LIN {X 0,Y 523.515,Z 542.317,A -85,B 0,C 180,E1 -4776.742,E2 -4776.742} C_VEL
LIN {X 0,Y 523.666,Z 535.608,A -85,B 0,C 180,E1 -4777.907,E2 -4777.907} C_VEL
LIN {X 0,Y 523.85,Z 527.307,A -85,B 0,C 180,E1 -4779.07,E2 -4779.07} C_VEL
LIN {X 0,Y 524.067,Z 518.801,A -85,B 0,C 180,E1 -4780.04,E2 -4780.04} C_VEL
LIN {X 0,Y 524.36,Z 508.293,A -85,B 0,C 180,E1 -4781.011,E2 -4781.011} C_VEL
LIN {X 0,Y 524.681,Z 496.847,A -85,B 0,C 180,E1 -4781.859,E2 -4781.859} C_VEL
LIN {X 0,Y 524.929,Z 486.505,A -85,B 0,C 180,E1 -4782.468,E2 -4782.468} C_VEL
LIN {X 0,Y 525.138,Z 474.81,A -85,B 0,C 180,E1 -4783.003,E2 -4783.003} C_VEL
LIN {X 0,Y 525.391,Z 461.34,A -85,B 0,C 180,E1 -4783.44,E2 -4783.44} C_VEL
LIN {X 0,Y 525.559,Z 448.003,A -85,B 0,C 180,E1 -4783.706,E2 -4783.706} C_VEL
LIN {X 0,Y 525.857,Z 355.901,A -85,B 0,C 180,E1 -4784.97,E2 -4784.97} C_VEL
LIN {X 0,Y 524.303,Z 345.51,A -85,B 0,C 180,E1 -4785.176,E2 -4785.176} C_VEL
LIN {X 0,Y 524.737,Z 323.457,A -85,B 0,C 180,E1 -4788.528,E2 -4788.528} C_VEL
LIN {X 0,Y 525.117,Z 304.861,A -85,B 0,C 180,E1 -4791.39,E2 -4791.39} C_VEL
LIN {X 0,Y 525.357,Z 292.969,A -85,B 0,C 180,E1 -4793.243,E2 -4793.243} C_VEL
LIN {X 0,Y 523.98,Z 285.215,A -85,B 0,C 180,E1 -4794.569,E2 -4794.569} C_VEL
LIN {X 0,Y 523.949,Z 285.218,A -85,B 0,C 180,E1 -4797.133,E2 -4797.133} C_VEL
LIN {X 0,Y 523.944,Z 285.223,A -85,B 0,C 180,E1 -4799.756,E2 -4799.756} C_VEL
LIN {X 0,Y 523.935,Z 285.221,A -85,B 0,C 180,E1 -4802.449,E2 -4802.449} C_VEL
LIN {X 0,Y 523.921,Z 285.218,A -85,B 0,C 180,E1 -4805.227,E2 -4805.227} C_VEL
LIN {X 0,Y 523.917,Z 285.225,A -85,B 0,C 180,E1 -4808.102,E2 -4808.102} C_VEL
LIN {X 0,Y 523.94,Z 285.217,A -85,B 0,C 180,E1 -4811.092,E2 -4811.092} C_VEL
LIN {X 0,Y 523.931,Z 285.221,A -85,B 0,C 180,E1 -4814.229,E2 -4814.229} C_VEL
LIN {X 0,Y 523.917,Z 285.225,A -85,B 0,C 180,E1 -4816.832,E2 -4816.832} C_VEL
LIN {X 0,Y 523.939,Z 285.221,A -85,B 0,C 180,E1 -4818.907,E2 -4818.907} C_VEL
LIN {X 0,Y 523.915,Z 285.218,A -85,B 0,C 180,E1 -4821.898,E2 -4821.898} C_VEL
LIN {X 0,Y 523.924,Z 285.226,A -85,B 0,C 180,E1 -4824.911,E2 -4824.911} C_VEL
LIN {X 0,Y 523.934,Z 285.217,A -85,B 0,C 180,E1 -4827.679,E2 -4827.679} C_VEL
LIN {X 0,Y 523.953,Z 285.216,A -85,B 0,C 180,E1 -4830.676,E2 -4830.676} C_VEL
LIN {X 0,Y 523.973,Z 285.213,A -85,B 0,C 180,E1 -4833.728,E2 -4833.728} C_VEL
LIN {X 0,Y 523.925,Z 285.216,A -85,B 0,C 180,E1 -4836.27,E2 -4836.27} C_VEL
LIN {X 0,Y 523.945,Z 285.216,A -85,B 0,C 180,E1 -4838.766,E2 -4838.766} C_VEL
LIN {X 0,Y 523.95,Z 285.22,A -85,B 0,C 180,E1 -4841.221,E2 -4841.221} C_VEL
LIN {X 0,Y 523.936,Z 285.222,A -85,B 0,C 180,E1 -4843.639,E2 -4843.639} C_VEL
LIN {X 0,Y 523.942,Z 285.216,A -85,B 0,C 180,E1 -4846.028,E2 -4846.028} C_VEL
LIN {X 0,Y 524.011,Z 285.206,A -85,B 0,C 180,E1 -4848.394,E2 -4848.394} C_VEL
LIN {X 0,Y 524.001,Z 285.211,A -85,B 0,C 180,E1 -4851.516,E2 -4851.516} C_VEL
LIN {X 0,Y 524.079,Z 285.195,A -85,B 0,C 180,E1 -4854.614,E2 -4854.614} C_VEL
LIN {X 0,Y 524.11,Z 285.198,A -85,B 0,C 180,E1 -4857.694,E2 -4857.694} C_VEL
LIN {X 0,Y 524.12,Z 285.192,A -85,B 0,C 180,E1 -4860.768,E2 -4860.768} C_VEL
LIN {X 0,Y 524.07,Z 285.195,A -85,B 0,C 180,E1 -4863.075,E2 -4863.075} C_VEL
LIN {X 0,Y 524.035,Z 285.211,A -85,B 0,C 180,E1 -4866.159,E2 -4866.159} C_VEL
LIN {X 0,Y 524.001,Z 285.213,A -85,B 0,C 180,E1 -4868.484,E2 -4868.484} C_VEL
LIN {X 0,Y 524,Z 285.207,A -85,B 0,C 180,E1 -4871.739,E2 -4871.739} C_VEL
LIN {X 0,Y 523.992,Z 285.21,A -85,B 0,C 180,E1 -4875.053,E2 -4875.053} C_VEL
LIN {X 0,Y 523.962,Z 285.213,A -85,B 0,C 180,E1 -4877.969,E2 -4877.969} C_VEL
LIN {X 0,Y 523.97,Z 285.217,A -85,B 0,C 180,E1 -4880.41,E2 -4880.41} C_VEL
LIN {X 0,Y 523.915,Z 285.225,A -85,B 0,C 180,E1 -4882.893,E2 -4882.893} C_VEL
LIN {X 0,Y 523.951,Z 285.215,A -85,B 0,C 180,E1 -4885.419,E2 -4885.419} C_VEL
LIN {X 0,Y 523.966,Z 285.21,A -85,B 0,C 180,E1 -4887.999,E2 -4887.999} C_VEL
LIN {X 0,Y 523.943,Z 285.222,A -85,B 0,C 180,E1 -4890.855,E2 -4890.855} C_VEL
LIN {X 0,Y 523.957,Z 285.213,A -85,B 0,C 180,E1 -4893.735,E2 -4893.735} C_VEL
LIN {X 0,Y 523.902,Z 285.22,A -85,B 0,C 180,E1 -4896.401,E2 -4896.401} C_VEL
LIN {X 0,Y 523.919,Z 285.225,A -85,B 0,C 180,E1 -4899.085,E2 -4899.085} C_VEL
LIN {X 0,Y 523.951,Z 285.214,A -85,B 0,C 180,E1 -4902.119,E2 -4902.119} C_VEL
LIN {X 0,Y 523.941,Z 285.223,A -85,B 0,C 180,E1 -4905.31,E2 -4905.31} C_VEL
LIN {X 0,Y 523.914,Z 285.22,A -85,B 0,C 180,E1 -4906.905,E2 -4906.905} C_VEL
LIN {X 0,Y 523.25,Z 285.311,A -85,B 0,C 180,E1 -4907.546,E2 -4907.546} C_VEL
LIN {X 0,Y 520.41,Z 285.663,A -85,B 0,C 180,E1 -4908.588,E2 -4908.588} C_VEL
LIN {X 0,Y 518.006,Z 285.962,A -85,B 0,C 180,E1 -4909.427,E2 -4909.427} C_VEL
LIN {X 0,Y 516.969,Z 286.088,A -85,B 0,C 180,E1 -4910.075,E2 -4910.075} C_VEL
LIN {X 0,Y 516.881,Z 286.097,A -85,B 0,C 180,E1 -4910.294,E2 -4910.294} C_VEL
LIN {X 0,Y 516.877,Z 286.1,A -85,B 0,C 180,E1 -4913.343,E2 -4913.343} C_VEL
LIN {X 0,Y 516.907,Z 286.098,A -85,B 0,C 180,E1 -4916.121,E2 -4916.121} C_VEL
LIN {X 0,Y 516.892,Z 286.097,A -85,B 0,C 180,E1 -4918.936,E2 -4918.936} C_VEL
LIN {X 0,Y 516.971,Z 286.237,A -85,B 0,C 180,E1 -4920.438,E2 -4920.438} C_VEL
LIN {X 0,Y 517.368,Z 291.344,A -85,B 0,C 180,E1 -4921.39,E2 -4921.39} C_VEL
LIN {X 0,Y 517.217,Z 308.839,A -85,B 0,C 180,E1 -4924.604,E2 -4924.604} C_VEL
LIN {X 0,Y 517.184,Z 309.29,A -85,B 0,C 180,E1 -4924.685,E2 -4924.685} C_VEL
LIN {X 0,Y 519.153,Z 320.399,A -85,B 0,C 180,E1 -4924.906,E2 -4924.906} C_VEL
LIN {X 0,Y 518.582,Z 416.061,A -85,B 0,C 180,E1 -4926.249,E2 -4926.249} C_VEL
LIN {X 0,Y 518.424,Z 429.105,A -85,B 0,C 180,E1 -4926.586,E2 -4926.586} C_VEL
LIN {X 0,Y 518.222,Z 441.25,A -85,B 0,C 180,E1 -4927.051,E2 -4927.051} C_VEL
LIN {X 0,Y 517.957,Z 453.258,A -85,B 0,C 180,E1 -4927.671,E2 -4927.671} C_VEL
LIN {X 0,Y 517.642,Z 464.025,A -85,B 0,C 180,E1 -4928.391,E2 -4928.391} C_VEL
LIN {X 0,Y 517.359,Z 475.056,A -85,B 0,C 180,E1 -4929.317,E2 -4929.317} C_VEL
LIN {X 0,Y 517.034,Z 484.878,A -85,B 0,C 180,E1 -4930.341,E2 -4930.341} C_VEL
LIN {X 0,Y 516.799,Z 494.224,A -85,B 0,C 180,E1 -4931.568,E2 -4931.568} C_VEL
LIN {X 0,Y 516.605,Z 501.678,A -85,B 0,C 180,E1 -4932.789,E2 -4932.789} C_VEL
LIN {X 0,Y 516.447,Z 506.653,A -85,B 0,C 180,E1 -4933.801,E2 -4933.801} C_VEL
LIN {X 0,Y 516.405,Z 511.668,A -85,B 0,C 180,E1 -4935.077,E2 -4935.077} C_VEL
LIN {X 0,Y 516.31,Z 515.051,A -85,B 0,C 180,E1 -4936.219,E2 -4936.219} C_VEL
LIN {X 0,Y 516.23,Z 517.598,A -85,B 0,C 180,E1 -4937.418,E2 -4937.418} C_VEL
LIN {X 0,Y 516.282,Z 519.102,A -85,B 0,C 180,E1 -4938.555,E2 -4938.555} C_VEL
LIN {X 0,Y 516.238,Z 519.799,A -85,B 0,C 180,E1 -4939.806,E2 -4939.806} C_VEL
LIN {X 0,Y 516.176,Z 519.736,A -85,B 0,C 180,E1 -4940.596,E2 -4940.596} C_VEL
LIN {X 0,Y 516.213,Z 519.25,A -85,B 0,C 180,E1 -4941.387,E2 -4941.387} C_VEL
LIN {X 0,Y 516.267,Z 518.344,A -85,B 0,C 180,E1 -4942.176,E2 -4942.176} C_VEL
LIN {X 0,Y 516.37,Z 515.929,A -85,B 0,C 180,E1 -4943.494,E2 -4943.494} C_VEL
LIN {X 0,Y 516.315,Z 511.958,A -85,B 0,C 180,E1 -4944.924,E2 -4944.924} C_VEL
LIN {X 0,Y 516.425,Z 507.49,A -85,B 0,C 180,E1 -4946.098,E2 -4946.098} C_VEL
LIN {X 0,Y 516.568,Z 500.737,A -85,B 0,C 180,E1 -4947.465,E2 -4947.465} C_VEL
LIN {X 0,Y 516.788,Z 493.426,A -85,B 0,C 180,E1 -4948.636,E2 -4948.636} C_VEL
LIN {X 0,Y 517.068,Z 484.361,A -85,B 0,C 180,E1 -4949.805,E2 -4949.805} C_VEL
LIN {X 0,Y 517.273,Z 473.947,A -85,B 0,C 180,E1 -4950.875,E2 -4950.875} C_VEL
LIN {X 0,Y 517.65,Z 463.329,A -85,B 0,C 180,E1 -4951.75,E2 -4951.75} C_VEL
LIN {X 0,Y 517.952,Z 453.041,A -85,B 0,C 180,E1 -4952.43,E2 -4952.43} C_VEL
LIN {X 0,Y 518.208,Z 440.744,A -85,B 0,C 180,E1 -4953.061,E2 -4953.061} C_VEL
LIN {X 0,Y 518.409,Z 427.821,A -85,B 0,C 180,E1 -4953.546,E2 -4953.546} C_VEL
LIN {X 0,Y 518.626,Z 414.887,A -85,B 0,C 180,E1 -4953.86,E2 -4953.86} C_VEL
LIN {X 0,Y 519.096,Z 319.758,A -85,B 0,C 180,E1 -4955.194,E2 -4955.194} C_VEL
LIN {X 0,Y 517.207,Z 309.344,A -85,B 0,C 180,E1 -4955.409,E2 -4955.409} C_VEL
LIN {X 0,Y 517.397,Z 294.542,A -85,B 0,C 180,E1 -4958.199,E2 -4958.199} C_VEL
LIN {X 0,Y 517.281,Z 288.307,A -85,B 0,C 180,E1 -4959.383,E2 -4959.383} C_VEL
LIN {X 0,Y 516.903,Z 286.101,A -85,B 0,C 180,E1 -4959.834,E2 -4959.834} C_VEL
LIN {X 0,Y 516.898,Z 286.099,A -85,B 0,C 180,E1 -4962.564,E2 -4962.564} C_VEL
LIN {X 0,Y 516.883,Z 286.096,A -85,B 0,C 180,E1 -4965.779,E2 -4965.779} C_VEL
LIN {X 0,Y 516.87,Z 286.102,A -85,B 0,C 180,E1 -4968.223,E2 -4968.223} C_VEL
LIN {X 0,Y 516.9,Z 286.098,A -85,B 0,C 180,E1 -4970.701,E2 -4970.701} C_VEL
LIN {X 0,Y 516.854,Z 286.098,A -85,B 0,C 180,E1 -4973.223,E2 -4973.223} C_VEL
LIN {X 0,Y 516.865,Z 286.099,A -85,B 0,C 180,E1 -4976.178,E2 -4976.178} C_VEL
LIN {X 0,Y 516.899,Z 286.093,A -85,B 0,C 180,E1 -4979.305,E2 -4979.305} C_VEL
LIN {X 0,Y 516.887,Z 286.099,A -85,B 0,C 180,E1 -4982.542,E2 -4982.542} C_VEL
LIN {X 0,Y 516.86,Z 286.099,A -85,B 0,C 180,E1 -4985.329,E2 -4985.329} C_VEL
LIN {X 0,Y 516.873,Z 286.095,A -85,B 0,C 180,E1 -4987.942,E2 -4987.942} C_VEL
LIN {X 0,Y 516.848,Z 286.104,A -85,B 0,C 180,E1 -4990.744,E2 -4990.744} C_VEL
LIN {X 0,Y 516.875,Z 286.095,A -85,B 0,C 180,E1 -4993.903,E2 -4993.903} C_VEL
LIN {X 0,Y 516.874,Z 286.095,A -85,B 0,C 180,E1 -4996.107,E2 -4996.107} C_VEL
LIN {X 0,Y 516.873,Z 286.105,A -85,B 0,C 180,E1 -4999.257,E2 -4999.257} C_VEL
LIN {X 0,Y 516.855,Z 286.097,A -85,B 0,C 180,E1 -5002.273,E2 -5002.273} C_VEL
LIN {X 0,Y 516.875,Z 286.101,A -85,B 0,C 180,E1 -5005.175,E2 -5005.175} C_VEL
LIN {X 0,Y 516.865,Z 286.098,A -85,B 0,C 180,E1 -5007.975,E2 -5007.975} C_VEL
LIN {X 0,Y 516.912,Z 286.09,A -85,B 0,C 180,E1 -5010.695,E2 -5010.695} C_VEL
LIN {X 0,Y 516.931,Z 286.095,A -85,B 0,C 180,E1 -5013.804,E2 -5013.804} C_VEL
LIN {X 0,Y 516.851,Z 286.098,A -85,B 0,C 180,E1 -5016.776,E2 -5016.776} C_VEL
LIN {X 0,Y 516.93,Z 286.097,A -85,B 0,C 180,E1 -5019.731,E2 -5019.731} C_VEL
LIN {X 0,Y 516.92,Z 286.09,A -85,B 0,C 180,E1 -5022.596,E2 -5022.596} C_VEL
LIN {X 0,Y 516.931,Z 286.088,A -85,B 0,C 180,E1 -5025.03,E2 -5025.03} C_VEL
LIN {X 0,Y 516.956,Z 286.091,A -85,B 0,C 180,E1 -5028.234,E2 -5028.234} C_VEL
LIN {X 0,Y 516.959,Z 286.085,A -85,B 0,C 180,E1 -5031.4,E2 -5031.4} C_VEL
LIN {X 0,Y 517.016,Z 286.081,A -85,B 0,C 180,E1 -5034.54,E2 -5034.54} C_VEL
LIN {X 0,Y 517.073,Z 286.072,A -85,B 0,C 180,E1 -5037.663,E2 -5037.663} C_VEL
LIN {X 0,Y 517.086,Z 286.072,A -85,B 0,C 180,E1 -5040.779,E2 -5040.779} C_VEL
LIN {X 0,Y 517.006,Z 286.079,A -85,B 0,C 180,E1 -5043.117,E2 -5043.117} C_VEL
LIN {X 0,Y 517,Z 286.085,A -85,B 0,C 180,E1 -5046.243,E2 -5046.243} C_VEL
LIN {X 0,Y 516.949,Z 286.086,A -85,B 0,C 180,E1 -5049.389,E2 -5049.389} C_VEL
LIN {X 0,Y 516.949,Z 286.086,A -85,B 0,C 180,E1 -5051.81,E2 -5051.81} C_VEL
LIN {X 0,Y 516.938,Z 286.09,A -85,B 0,C 180,E1 -5055.148,E2 -5055.148} C_VEL
LIN {X 0,Y 516.917,Z 286.091,A -85,B 0,C 180,E1 -5058.223,E2 -5058.223} C_VEL
LIN {X 0,Y 516.904,Z 286.098,A -85,B 0,C 180,E1 -5060.702,E2 -5060.702} C_VEL
LIN {X 0,Y 516.904,Z 286.091,A -85,B 0,C 180,E1 -5064.073,E2 -5064.073} C_VEL
LIN {X 0,Y 516.922,Z 286.093,A -85,B 0,C 180,E1 -5066.658,E2 -5066.658} C_VEL
LIN {X 0,Y 516.913,Z 286.093,A -85,B 0,C 180,E1 -5069.526,E2 -5069.526} C_VEL
LIN {X 0,Y 516.894,Z 286.094,A -85,B 0,C 180,E1 -5072.545,E2 -5072.545} C_VEL
LIN {X 0,Y 516.873,Z 286.104,A -85,B 0,C 180,E1 -5075.333,E2 -5075.333} C_VEL
LIN {X 0,Y 516.879,Z 286.096,A -85,B 0,C 180,E1 -5077.944,E2 -5077.944} C_VEL
LIN {X 0,Y 516.881,Z 286.095,A -85,B 0,C 180,E1 -5080.742,E2 -5080.742} C_VEL
LIN {X 0,Y 516.9,Z 286.093,A -85,B 0,C 180,E1 -5082.83,E2 -5082.83} C_VEL
LIN {X 0,Y 516.919,Z 286.092,A -85,B 0,C 180,E1 -5085.011,E2 -5085.011} C_VEL
LIN {X 0,Y 516.912,Z 286.091,A -85,B 0,C 180,E1 -5088.399,E2 -5088.399} C_VEL
LIN {X 0,Y 516.877,Z 286.098,A -85,B 0,C 180,E1 -5091.285,E2 -5091.285} C_VEL
LIN {X 0,Y 516.869,Z 286.099,A -85,B 0,C 180,E1 -5094.221,E2 -5094.221} C_VEL
LIN {X 0,Y 516.893,Z 286.093,A -85,B 0,C 180,E1 -5097.054,E2 -5097.054} C_VEL
LIN {X 0,Y 516.891,Z 286.101,A -85,B 0,C 180,E1 -5099.797,E2 -5099.797} C_VEL
LIN {X 0,Y 516.928,Z 286.093,A -85,B 0,C 180,E1 -5102.468,E2 -5102.468} C_VEL
LIN {X 0,Y 516.974,Z 286.201,A -85,B 0,C 180,E1 -5105.275,E2 -5105.275} C_VEL
LIN {X 0,Y 518.519,Z 295.613,A -85,B 0,C 180,E1 -5106.855,E2 -5106.855} C_VEL
LIN {X 0,Y 517.945,Z 316.638,A -85,B 0,C 180,E1 -5110.171,E2 -5110.171} C_VEL
LIN {X 0,Y 517.417,Z 336.293,A -85,B 0,C 180,E1 -5113.224,E2 -5113.224} C_VEL
LIN {X 0,Y 517.289,Z 345.545,A -85,B 0,C 180,E1 -5114.634,E2 -5114.634} C_VEL
LIN {X 0,Y 519.035,Z 357.742,A -85,B 0,C 180,E1 -5114.857,E2 -5114.857} C_VEL
LIN {X 0,Y 518.607,Z 453.704,A -85,B 0,C 180,E1 -5116.207,E2 -5116.207} C_VEL
LIN {X 0,Y 518.362,Z 466.254,A -85,B 0,C 180,E1 -5116.525,E2 -5116.525} C_VEL
LIN {X 0,Y 518.098,Z 479.211,A -85,B 0,C 180,E1 -5117.017,E2 -5117.017} C_VEL
LIN {X 0,Y 517.831,Z 491.38,A -85,B 0,C 180,E1 -5117.649,E2 -5117.649} C_VEL
LIN {X 0,Y 517.517,Z 503.136,A -85,B 0,C 180,E1 -5118.446,E2 -5118.446} C_VEL
LIN {X 0,Y 517.215,Z 513.599,A -85,B 0,C 180,E1 -5119.331,E2 -5119.331} C_VEL
LIN {X 0,Y 516.958,Z 522.155,A -85,B 0,C 180,E1 -5120.216,E2 -5120.216} C_VEL
LIN {X 0,Y 516.723,Z 530.05,A -85,B 0,C 180,E1 -5121.199,E2 -5121.199} C_VEL
LIN {X 0,Y 516.544,Z 537.763,A -85,B 0,C 180,E1 -5122.377,E2 -5122.377} C_VEL
LIN {X 0,Y 516.395,Z 544.873,A -85,B 0,C 180,E1 -5123.75,E2 -5123.75} C_VEL
LIN {X 0,Y 516.313,Z 549.603,A -85,B 0,C 180,E1 -5124.924,E2 -5124.924} C_VEL
LIN {X 0,Y 516.352,Z 553.22,A -85,B 0,C 180,E1 -5126.098,E2 -5126.098} C_VEL
LIN {X 0,Y 516.282,Z 555.082,A -85,B 0,C 180,E1 -5126.879,E2 -5126.879} C_VEL
LIN {X 0,Y 516.26,Z 556.48,A -85,B 0,C 180,E1 -5127.66,E2 -5127.66} C_VEL
LIN {X 0,Y 516.16,Z 558.081,A -85,B 0,C 180,E1 -5129.22,E2 -5129.22} C_VEL
LIN {X 0,Y 516.158,Z 558.297,A -85,B 0,C 180,E1 -5130,E2 -5130} C_VEL
LIN {X 0,Y 516.191,Z 557.472,A -85,B 0,C 180,E1 -5131.561,E2 -5131.561} C_VEL
LIN {X 0,Y 516.261,Z 556.476,A -85,B 0,C 180,E1 -5132.341,E2 -5132.341} C_VEL
LIN {X 0,Y 516.282,Z 555.077,A -85,B 0,C 180,E1 -5133.122,E2 -5133.122} C_VEL
LIN {X 0,Y 516.312,Z 552.135,A -85,B 0,C 180,E1 -5134.294,E2 -5134.294} C_VEL
LIN {X 0,Y 516.376,Z 548.153,A -85,B 0,C 180,E1 -5135.467,E2 -5135.467} C_VEL
LIN {X 0,Y 516.422,Z 542.93,A -85,B 0,C 180,E1 -5136.663,E2 -5136.663} C_VEL
LIN {X 0,Y 516.581,Z 536.576,A -85,B 0,C 180,E1 -5137.82,E2 -5137.82} C_VEL
LIN {X 0,Y 516.769,Z 528.529,A -85,B 0,C 180,E1 -5138.998,E2 -5138.998} C_VEL
LIN {X 0,Y 516.988,Z 520.331,A -85,B 0,C 180,E1 -5139.981,E2 -5139.981} C_VEL
LIN {X 0,Y 517.285,Z 510.336,A -85,B 0,C 180,E1 -5140.965,E2 -5140.965} C_VEL
LIN {X 0,Y 517.603,Z 500.479,A -85,B 0,C 180,E1 -5141.752,E2 -5141.752} C_VEL
LIN {X 0,Y 517.864,Z 489.277,A -85,B 0,C 180,E1 -5142.469,E2 -5142.469} C_VEL
LIN {X 0,Y 518.138,Z 476.878,A -85,B 0,C 180,E1 -5143.082,E2 -5143.082} C_VEL
LIN {X 0,Y 518.418,Z 463.797,A -85,B 0,C 180,E1 -5143.549,E2 -5143.549} C_VEL
LIN {X 0,Y 518.643,Z 450.736,A -85,B 0,C 180,E1 -5143.843,E2 -5143.843} C_VEL
LIN {X 0,Y 518.935,Z 356.179,A -85,B 0,C 180,E1 -5145.167,E2 -5145.167} C_VEL
LIN {X 0,Y 517.272,Z 345.308,A -85,B 0,C 180,E1 -5145.376,E2 -5145.376} C_VEL
LIN {X 0,Y 517.742,Z 324.36,A -85,B 0,C 180,E1 -5148.602,E2 -5148.602} C_VEL
LIN {X 0,Y 518.167,Z 305.904,A -85,B 0,C 180,E1 -5151.482,E2 -5151.482} C_VEL
LIN {X 0,Y 518.39,Z 294.032,A -85,B 0,C 180,E1 -5153.363,E2 -5153.363} C_VEL
LIN {X 0,Y 516.932,Z 286.093,A -85,B 0,C 180,E1 -5154.742,E2 -5154.742} C_VEL
LIN {X 0,Y 516.926,Z 286.096,A -85,B 0,C 180,E1 -5157.533,E2 -5157.533} C_VEL
LIN {X 0,Y 516.894,Z 286.102,A -85,B 0,C 180,E1 -5160.204,E2 -5160.204} C_VEL
LIN {X 0,Y 516.896,Z 286.093,A -85,B 0,C 180,E1 -5162.947,E2 -5162.947} C_VEL
LIN {X 0,Y 516.873,Z 286.099,A -85,B 0,C 180,E1 -5165.78,E2 -5165.78} C_VEL
LIN {X 0,Y 516.881,Z 286.1,A -85,B 0,C 180,E1 -5168.716,E2 -5168.716} C_VEL
LIN {X 0,Y 516.912,Z 286.092,A -85,B 0,C 180,E1 -5171.775,E2 -5171.775} C_VEL
LIN {X 0,Y 516.895,Z 286.097,A -85,B 0,C 180,E1 -5175.007,E2 -5175.007} C_VEL
LIN {X 0,Y 516.913,Z 286.095,A -85,B 0,C 180,E1 -5178.399,E2 -5178.399} C_VEL
LIN {X 0,Y 516.88,Z 286.097,A -85,B 0,C 180,E1 -5181.284,E2 -5181.284} C_VEL
LIN {X 0,Y 516.87,Z 286.096,A -85,B 0,C 180,E1 -5184.219,E2 -5184.219} C_VEL
LIN {X 0,Y 516.894,Z 286.102,A -85,B 0,C 180,E1 -5187.053,E2 -5187.053} C_VEL
LIN {X 0,Y 516.891,Z 286.093,A -85,B 0,C 180,E1 -5189.796,E2 -5189.796} C_VEL
LIN {X 0,Y 516.925,Z 286.09,A -85,B 0,C 180,E1 -5192.467,E2 -5192.467} C_VEL
LIN {X 0,Y 516.908,Z 286.098,A -85,B 0,C 180,E1 -5195.072,E2 -5195.072} C_VEL
LIN {X 0,Y 516.884,Z 286.094,A -85,B 0,C 180,E1 -5198.462,E2 -5198.462} C_VEL
LIN {X 0,Y 516.902,Z 286.094,A -85,B 0,C 180,E1 -5200.955,E2 -5200.955} C_VEL
LIN {X 0,Y 516.912,Z 286.098,A -85,B 0,C 180,E1 -5203.41,E2 -5203.41} C_VEL
LIN {X 0,Y 516.904,Z 286.095,A -85,B 0,C 180,E1 -5205.834,E2 -5205.834} C_VEL
LIN {X 0,Y 516.949,Z 286.086,A -85,B 0,C 180,E1 -5209.028,E2 -5209.028} C_VEL
LIN {X 0,Y 516.976,Z 286.084,A -85,B 0,C 180,E1 -5212.187,E2 -5212.187} C_VEL
LIN {X 0,Y 517.026,Z 286.074,A -85,B 0,C 180,E1 -5214.54,E2 -5214.54} C_VEL
LIN {X 0,Y 517.082,Z 286.073,A -85,B 0,C 180,E1 -5217.663,E2 -5217.663} C_VEL
LIN {X 0,Y 517.09,Z 286.067,A -85,B 0,C 180,E1 -5220.779,E2 -5220.779} C_VEL
LIN {X 0,Y 517.011,Z 286.075,A -85,B 0,C 180,E1 -5223.117,E2 -5223.117} C_VEL
LIN {X 0,Y 517,Z 286.087,A -85,B 0,C 180,E1 -5226.243,E2 -5226.243} C_VEL
LIN {X 0,Y 516.949,Z 286.085,A -85,B 0,C 180,E1 -5229.389,E2 -5229.389} C_VEL
LIN {X 0,Y 516.95,Z 286.086,A -85,B 0,C 180,E1 -5231.807,E2 -5231.807} C_VEL
LIN {X 0,Y 516.945,Z 286.087,A -85,B 0,C 180,E1 -5235.147,E2 -5235.147} C_VEL
LIN {X 0,Y 516.923,Z 286.093,A -85,B 0,C 180,E1 -5238.222,E2 -5238.222} C_VEL
LIN {X 0,Y 516.911,Z 286.098,A -85,B 0,C 180,E1 -5240.701,E2 -5240.701} C_VEL
LIN {X 0,Y 516.91,Z 286.091,A -85,B 0,C 180,E1 -5244.072,E2 -5244.072} C_VEL
LIN {X 0,Y 516.923,Z 286.095,A -85,B 0,C 180,E1 -5246.658,E2 -5246.658} C_VEL
LIN {X 0,Y 516.909,Z 286.092,A -85,B 0,C 180,E1 -5249.524,E2 -5249.524} C_VEL
LIN {X 0,Y 516.894,Z 286.094,A -85,B 0,C 180,E1 -5252.543,E2 -5252.543} C_VEL
LIN {X 0,Y 516.865,Z 286.103,A -85,B 0,C 180,E1 -5255.33,E2 -5255.33} C_VEL
LIN {X 0,Y 516.879,Z 286.095,A -85,B 0,C 180,E1 -5257.943,E2 -5257.943} C_VEL
LIN {X 0,Y 516.882,Z 286.095,A -85,B 0,C 180,E1 -5260.742,E2 -5260.742} C_VEL
LIN {X 0,Y 516.881,Z 286.097,A -85,B 0,C 180,E1 -5262.832,E2 -5262.832} C_VEL
LIN {X 0,Y 516.894,Z 286.097,A -85,B 0,C 180,E1 -5265.007,E2 -5265.007} C_VEL
LIN {X 0,Y 516.913,Z 286.091,A -85,B 0,C 180,E1 -5268.399,E2 -5268.399} C_VEL
LIN {X 0,Y 516.881,Z 286.097,A -85,B 0,C 180,E1 -5270.294,E2 -5270.294} C_VEL
LIN {X 0,Y 516.209,Z 286.181,A -85,B 0,C 180,E1 -5270.944,E2 -5270.944} C_VEL
LIN {X 0,Y 513.363,Z 286.544,A -85,B 0,C 180,E1 -5272,E2 -5272} C_VEL
LIN {X 0,Y 510.954,Z 286.848,A -85,B 0,C 180,E1 -5272.85,E2 -5272.85} C_VEL
LIN {X 0,Y 509.911,Z 286.975,A -85,B 0,C 180,E1 -5273.506,E2 -5273.506} C_VEL
LIN {X 0,Y 509.821,Z 286.983,A -85,B 0,C 180,E1 -5273.729,E2 -5273.729} C_VEL
LIN {X 0,Y 509.859,Z 286.973,A -85,B 0,C 180,E1 -5276.539,E2 -5276.539} C_VEL
LIN {X 0,Y 509.853,Z 286.977,A -85,B 0,C 180,E1 -5279.335,E2 -5279.335} C_VEL
LIN {X 0,Y 509.922,Z 287.05,A -85,B 0,C 180,E1 -5280.297,E2 -5280.297} C_VEL
LIN {X 0,Y 510.408,Z 291.735,A -85,B 0,C 180,E1 -5281.189,E2 -5281.189} C_VEL
LIN {X 0,Y 510.227,Z 308.501,A -85,B 0,C 180,E1 -5284.285,E2 -5284.285} C_VEL
LIN {X 0,Y 510.237,Z 309.421,A -85,B 0,C 180,E1 -5284.456,E2 -5284.456} C_VEL
LIN {X 0,Y 512.335,Z 321.922,A -85,B 0,C 180,E1 -5284.717,E2 -5284.717} C_VEL
LIN {X 0,Y 511.702,Z 416.819,A -85,B 0,C 180,E1 -5286.071,E2 -5286.071} C_VEL
LIN {X 0,Y 511.487,Z 430.471,A -85,B 0,C 180,E1 -5286.437,E2 -5286.437} C_VEL
LIN {X 0,Y 511.275,Z 442.481,A -85,B 0,C 180,E1 -5286.915,E2 -5286.915} C_VEL
LIN {X 0,Y 511.007,Z 454.524,A -85,B 0,C 180,E1 -5287.564,E2 -5287.564} C_VEL
LIN {X 0,Y 510.606,Z 466.435,A -85,B 0,C 180,E1 -5288.396,E2 -5288.396} C_VEL
LIN {X 0,Y 510.318,Z 476.796,A -85,B 0,C 180,E1 -5289.308,E2 -5289.308} C_VEL
LIN {X 0,Y 510.005,Z 485.651,A -85,B 0,C 180,E1 -5290.268,E2 -5290.268} C_VEL
LIN {X 0,Y 509.791,Z 493.511,A -85,B 0,C 180,E1 -5291.305,E2 -5291.305} C_VEL
LIN {X 0,Y 509.553,Z 501.139,A -85,B 0,C 180,E1 -5292.543,E2 -5292.543} C_VEL
LIN {X 0,Y 509.403,Z 506.27,A -85,B 0,C 180,E1 -5293.571,E2 -5293.571} C_VEL
LIN {X 0,Y 509.309,Z 511.916,A -85,B 0,C 180,E1 -5295.002,E2 -5295.002} C_VEL
LIN {X 0,Y 509.183,Z 515.946,A -85,B 0,C 180,E1 -5296.429,E2 -5296.429} C_VEL
LIN {X 0,Y 509.152,Z 517.606,A -85,B 0,C 180,E1 -5297.241,E2 -5297.241} C_VEL
LIN {X 0,Y 509.185,Z 519.347,A -85,B 0,C 180,E1 -5298.514,E2 -5298.514} C_VEL
LIN {X 0,Y 509.157,Z 520.035,A -85,B 0,C 180,E1 -5299.662,E2 -5299.662} C_VEL
LIN {X 0,Y 509.12,Z 519.631,A -85,B 0,C 180,E1 -5301.266,E2 -5301.266} C_VEL
LIN {X 0,Y 509.17,Z 518.804,A -85,B 0,C 180,E1 -5302.066,E2 -5302.066} C_VEL
LIN {X 0,Y 509.287,Z 516.278,A -85,B 0,C 180,E1 -5303.503,E2 -5303.503} C_VEL
LIN {X 0,Y 509.244,Z 512.649,A -85,B 0,C 180,E1 -5304.853,E2 -5304.853} C_VEL
LIN {X 0,Y 509.351,Z 508.309,A -85,B 0,C 180,E1 -5306.044,E2 -5306.044} C_VEL
LIN {X 0,Y 509.489,Z 502.801,A -85,B 0,C 180,E1 -5307.232,E2 -5307.232} C_VEL
LIN {X 0,Y 509.648,Z 495.952,A -85,B 0,C 180,E1 -5308.419,E2 -5308.419} C_VEL
LIN {X 0,Y 509.951,Z 487.378,A -85,B 0,C 180,E1 -5309.605,E2 -5309.605} C_VEL
LIN {X 0,Y 510.179,Z 478.642,A -85,B 0,C 180,E1 -5310.592,E2 -5310.592} C_VEL
LIN {X 0,Y 510.493,Z 467.904,A -85,B 0,C 180,E1 -5311.577,E2 -5311.577} C_VEL
LIN {X 0,Y 510.922,Z 457.034,A -85,B 0,C 180,E1 -5312.365,E2 -5312.365} C_VEL
LIN {X 0,Y 511.242,Z 444.935,A -85,B 0,C 180,E1 -5313.053,E2 -5313.053} C_VEL
LIN {X 0,Y 511.509,Z 432.195,A -85,B 0,C 180,E1 -5313.594,E2 -5313.594} C_VEL
LIN {X 0,Y 511.698,Z 420.431,A -85,B 0,C 180,E1 -5313.937,E2 -5313.937} C_VEL
LIN {X 0,Y 511.836,Z 404.682,A -85,B 0,C 180,E1 -5314.207,E2 -5314.207} C_VEL
LIN {X 0,Y 512.23,Z 320.41,A -85,B 0,C 180,E1 -5315.397,E2 -5315.397} C_VEL
LIN {X 0,Y 510.186,Z 309.514,A -85,B 0,C 180,E1 -5315.632,E2 -5315.632} C_VEL
LIN {X 0,Y 510.425,Z 295.354,A -85,B 0,C 180,E1 -5318.312,E2 -5318.312} C_VEL
LIN {X 0,Y 510.263,Z 289.11,A -85,B 0,C 180,E1 -5319.513,E2 -5319.513} C_VEL
LIN {X 0,Y 509.835,Z 286.982,A -85,B 0,C 180,E1 -5319.972,E2 -5319.972} C_VEL
LIN {X 0,Y 509.859,Z 286.974,A -85,B 0,C 180,E1 -5322.741,E2 -5322.741} C_VEL
LIN {X 0,Y 509.894,Z 286.964,A -85,B 0,C 180,E1 -5325.241,E2 -5325.241} C_VEL
LIN {X 0,Y 509.828,Z 286.981,A -85,B 0,C 180,E1 -5328.484,E2 -5328.484} C_VEL
LIN {X 0,Y 509.843,Z 286.973,A -85,B 0,C 180,E1 -5331.001,E2 -5331.001} C_VEL
LIN {X 0,Y 509.815,Z 286.974,A -85,B 0,C 180,E1 -5333.563,E2 -5333.563} C_VEL
LIN {X 0,Y 509.804,Z 286.981,A -85,B 0,C 180,E1 -5336.354,E2 -5336.354} C_VEL
LIN {X 0,Y 509.832,Z 286.979,A -85,B 0,C 180,E1 -5338.846,E2 -5338.846} C_VEL
LIN {X 0,Y 509.808,Z 286.975,A -85,B 0,C 180,E1 -5341.59,E2 -5341.59} C_VEL
LIN {X 0,Y 509.833,Z 286.975,A -85,B 0,C 180,E1 -5344.414,E2 -5344.414} C_VEL
LIN {X 0,Y 509.811,Z 286.978,A -85,B 0,C 180,E1 -5347.34,E2 -5347.34} C_VEL
LIN {X 0,Y 509.808,Z 286.977,A -85,B 0,C 180,E1 -5350.384,E2 -5350.384} C_VEL
LIN {X 0,Y 509.794,Z 286.987,A -85,B 0,C 180,E1 -5353.059,E2 -5353.059} C_VEL
LIN {X 0,Y 509.815,Z 286.975,A -85,B 0,C 180,E1 -5355.793,E2 -5355.793} C_VEL
LIN {X 0,Y 509.844,Z 286.972,A -85,B 0,C 180,E1 -5358.573,E2 -5358.573} C_VEL
LIN {X 0,Y 509.842,Z 286.973,A -85,B 0,C 180,E1 -5361.786,E2 -5361.786} C_VEL
LIN {X 0,Y 509.822,Z 286.974,A -85,B 0,C 180,E1 -5364.621,E2 -5364.621} C_VEL
LIN {X 0,Y 509.853,Z 286.979,A -85,B 0,C 180,E1 -5367.48,E2 -5367.48} C_VEL
LIN {X 0,Y 509.85,Z 286.97,A -85,B 0,C 180,E1 -5370.273,E2 -5370.273} C_VEL
LIN {X 0,Y 509.865,Z 286.969,A -85,B 0,C 180,E1 -5372.943,E2 -5372.943} C_VEL
LIN {X 0,Y 509.842,Z 286.979,A -85,B 0,C 180,E1 -5375.573,E2 -5375.573} C_VEL
LIN {X 0,Y 509.812,Z 286.978,A -85,B 0,C 180,E1 -5378.148,E2 -5378.148} C_VEL
LIN {X 0,Y 509.854,Z 286.97,A -85,B 0,C 180,E1 -5380.681,E2 -5380.681} C_VEL
LIN {X 0,Y 509.874,Z 286.968,A -85,B 0,C 180,E1 -5383.174,E2 -5383.174} C_VEL
LIN {X 0,Y 509.852,Z 286.975,A -85,B 0,C 180,E1 -5385.634,E2 -5385.634} C_VEL
LIN {X 0,Y 509.904,Z 286.963,A -85,B 0,C 180,E1 -5388.874,E2 -5388.874} C_VEL
LIN {X 0,Y 509.942,Z 286.968,A -85,B 0,C 180,E1 -5392.078,E2 -5392.078} C_VEL
LIN {X 0,Y 509.966,Z 286.96,A -85,B 0,C 180,E1 -5394.464,E2 -5394.464} C_VEL
LIN {X 0,Y 510.044,Z 286.947,A -85,B 0,C 180,E1 -5397.631,E2 -5397.631} C_VEL
LIN {X 0,Y 510.056,Z 286.947,A -85,B 0,C 180,E1 -5400.79,E2 -5400.79} C_VEL
LIN {X 0,Y 509.948,Z 286.958,A -85,B 0,C 180,E1 -5403.16,E2 -5403.16} C_VEL
LIN {X 0,Y 509.969,Z 286.962,A -85,B 0,C 180,E1 -5406.33,E2 -5406.33} C_VEL
LIN {X 0,Y 509.91,Z 286.969,A -85,B 0,C 180,E1 -5408.72,E2 -5408.72} C_VEL
LIN {X 0,Y 509.897,Z 286.965,A -85,B 0,C 180,E1 -5411.932,E2 -5411.932} C_VEL
LIN {X 0,Y 509.885,Z 286.968,A -85,B 0,C 180,E1 -5415.242,E2 -5415.242} C_VEL
LIN {X 0,Y 509.88,Z 286.967,A -85,B 0,C 180,E1 -5418.001,E2 -5418.001} C_VEL
LIN {X 0,Y 509.842,Z 286.979,A -85,B 0,C 180,E1 -5421.002,E2 -5421.002} C_VEL
LIN {X 0,Y 509.863,Z 286.97,A -85,B 0,C 180,E1 -5424.426,E2 -5424.426} C_VEL
LIN {X 0,Y 509.88,Z 286.976,A -85,B 0,C 180,E1 -5427.056,E2 -5427.056} C_VEL
LIN {X 0,Y 509.874,Z 286.968,A -85,B 0,C 180,E1 -5429.75,E2 -5429.75} C_VEL
LIN {X 0,Y 509.87,Z 286.971,A -85,B 0,C 180,E1 -5432.776,E2 -5432.776} C_VEL
LIN {X 0,Y 509.833,Z 286.977,A -85,B 0,C 180,E1 -5435.581,E2 -5435.581} C_VEL
LIN {X 0,Y 509.846,Z 286.97,A -85,B 0,C 180,E1 -5438.339,E2 -5438.339} C_VEL
LIN {X 0,Y 509.854,Z 286.979,A -85,B 0,C 180,E1 -5441.426,E2 -5441.426} C_VEL
LIN {X 0,Y 509.852,Z 286.97,A -85,B 0,C 180,E1 -5444.669,E2 -5444.669} C_VEL
LIN {X 0,Y 509.854,Z 286.972,A -85,B 0,C 180,E1 -5448.104,E2 -5448.104} C_VEL
LIN {X 0,Y 509.842,Z 286.971,A -85,B 0,C 180,E1 -5450.648,E2 -5450.648} C_VEL
LIN {X 0,Y 509.822,Z 286.982,A -85,B 0,C 180,E1 -5453.648,E2 -5453.648} C_VEL
LIN {X 0,Y 509.857,Z 286.97,A -85,B 0,C 180,E1 -5456.54,E2 -5456.54} C_VEL
LIN {X 0,Y 509.844,Z 286.973,A -85,B 0,C 180,E1 -5459.335,E2 -5459.335} C_VEL
LIN {X 0,Y 509.894,Z 286.974,A -85,B 0,C 180,E1 -5462.055,E2 -5462.055} C_VEL
LIN {X 0,Y 509.904,Z 287.016,A -85,B 0,C 180,E1 -5465.099,E2 -5465.099} C_VEL
LIN {X 0,Y 511.443,Z 295.302,A -85,B 0,C 180,E1 -5466.516,E2 -5466.516} C_VEL
LIN {X 0,Y 511.301,Z 304.536,A -85,B 0,C 180,E1 -5468.004,E2 -5468.004} C_VEL
LIN {X 0,Y 510.807,Z 322.937,A -85,B 0,C 180,E1 -5470.928,E2 -5470.928} C_VEL
LIN {X 0,Y 510.33,Z 342.578,A -85,B 0,C 180,E1 -5474.013,E2 -5474.013} C_VEL
LIN {X 0,Y 510.273,Z 345.283,A -85,B 0,C 180,E1 -5474.417,E2 -5474.417} C_VEL
LIN {X 0,Y 512.169,Z 358.562,A -85,B 0,C 180,E1 -5474.665,E2 -5474.665} C_VEL
LIN {X 0,Y 511.711,Z 453.418,A -85,B 0,C 180,E1 -5476.017,E2 -5476.017} C_VEL
LIN {X 0,Y 511.442,Z 466.74,A -85,B 0,C 180,E1 -5476.365,E2 -5476.365} C_VEL
LIN {X 0,Y 511.165,Z 478.937,A -85,B 0,C 180,E1 -5476.838,E2 -5476.838} C_VEL
LIN {X 0,Y 510.919,Z 490.327,A -85,B 0,C 180,E1 -5477.432,E2 -5477.432} C_VEL
LIN {X 0,Y 510.545,Z 501.569,A -85,B 0,C 180,E1 -5478.185,E2 -5478.185} C_VEL
LIN {X 0,Y 510.252,Z 512.258,A -85,B 0,C 180,E1 -5479.084,E2 -5479.084} C_VEL
LIN {X 0,Y 509.922,Z 521.888,A -85,B 0,C 180,E1 -5480.08,E2 -5480.08} C_VEL
LIN {X 0,Y 509.671,Z 529.784,A -85,B 0,C 180,E1 -5481.076,E2 -5481.076} C_VEL
LIN {X 0,Y 509.479,Z 537.498,A -85,B 0,C 180,E1 -5482.271,E2 -5482.271} C_VEL
LIN {X 0,Y 509.308,Z 544.608,A -85,B 0,C 180,E1 -5483.663,E2 -5483.663} C_VEL
LIN {X 0,Y 509.243,Z 549.339,A -85,B 0,C 180,E1 -5484.854,E2 -5484.854} C_VEL
LIN {X 0,Y 509.245,Z 552.956,A -85,B 0,C 180,E1 -5486.044,E2 -5486.044} C_VEL
LIN {X 0,Y 509.2,Z 554.819,A -85,B 0,C 180,E1 -5486.836,E2 -5486.836} C_VEL
LIN {X 0,Y 509.189,Z 556.217,A -85,B 0,C 180,E1 -5487.627,E2 -5487.627} C_VEL
LIN {X 0,Y 509.073,Z 557.818,A -85,B 0,C 180,E1 -5489.209,E2 -5489.209} C_VEL
LIN {X 0,Y 509.069,Z 558.033,A -85,B 0,C 180,E1 -5490,E2 -5490} C_VEL
LIN {X 0,Y 509.112,Z 557.207,A -85,B 0,C 180,E1 -5491.582,E2 -5491.582} C_VEL
LIN {X 0,Y 509.189,Z 556.211,A -85,B 0,C 180,E1 -5492.374,E2 -5492.374} C_VEL
LIN {X 0,Y 509.2,Z 554.811,A -85,B 0,C 180,E1 -5493.165,E2 -5493.165} C_VEL
LIN {X 0,Y 509.204,Z 551.867,A -85,B 0,C 180,E1 -5494.354,E2 -5494.354} C_VEL
LIN {X 0,Y 509.293,Z 547.885,A -85,B 0,C 180,E1 -5495.544,E2 -5495.544} C_VEL
LIN {X 0,Y 509.4,Z 541.86,A -85,B 0,C 180,E1 -5496.914,E2 -5496.914} C_VEL
LIN {X 0,Y 509.545,Z 535.065,A -85,B 0,C 180,E1 -5498.128,E2 -5498.128} C_VEL
LIN {X 0,Y 509.748,Z 526.761,A -85,B 0,C 180,E1 -5499.323,E2 -5499.323} C_VEL
LIN {X 0,Y 510.012,Z 518.251,A -85,B 0,C 180,E1 -5500.32,E2 -5500.32} C_VEL
LIN {X 0,Y 510.389,Z 507.74,A -85,B 0,C 180,E1 -5501.316,E2 -5501.316} C_VEL
LIN {X 0,Y 510.709,Z 496.273,A -85,B 0,C 180,E1 -5502.19,E2 -5502.19} C_VEL
LIN {X 0,Y 511.013,Z 485.943,A -85,B 0,C 180,E1 -5502.813,E2 -5502.813} C_VEL
LIN {X 0,Y 511.281,Z 474.24,A -85,B 0,C 180,E1 -5503.362,E2 -5503.362} C_VEL
LIN {X 0,Y 511.56,Z 460.758,A -85,B 0,C 180,E1 -5503.81,E2 -5503.81} C_VEL
LIN {X 0,Y 511.772,Z 447.389,A -85,B 0,C 180,E1 -5504.083,E2 -5504.083} C_VEL
LIN {X 0,Y 512.109,Z 357.173,A -85,B 0,C 180,E1 -5505.356,E2 -5505.356} C_VEL
LIN {X 0,Y 510.237,Z 345.072,A -85,B 0,C 180,E1 -5505.587,E2 -5505.587} C_VEL
LIN {X 0,Y 510.751,Z 324.081,A -85,B 0,C 180,E1 -5508.867,E2 -5508.867} C_VEL
LIN {X 0,Y 511.226,Z 306.974,A -85,B 0,C 180,E1 -5511.577,E2 -5511.577} C_VEL
LIN {X 0,Y 511.558,Z 297.045,A -85,B 0,C 180,E1 -5513.168,E2 -5513.168} C_VEL
LIN {X 0,Y 510.475,Z 289.84,A -85,B 0,C 180,E1 -5514.395,E2 -5514.395} C_VEL
LIN {X 0,Y 509.89,Z 286.97,A -85,B 0,C 180,E1 -5514.899,E2 -5514.899} C_VEL
LIN {X 0,Y 509.884,Z 286.971,A -85,B 0,C 180,E1 -5517.056,E2 -5517.056} C_VEL
LIN {X 0,Y 509.86,Z 286.978,A -85,B 0,C 180,E1 -5519.751,E2 -5519.751} C_VEL
LIN {X 0,Y 509.875,Z 286.969,A -85,B 0,C 180,E1 -5522.774,E2 -5522.774} C_VEL
LIN {X 0,Y 509.827,Z 286.975,A -85,B 0,C 180,E1 -5525.578,E2 -5525.578} C_VEL
LIN {X 0,Y 509.851,Z 286.979,A -85,B 0,C 180,E1 -5528.338,E2 -5528.338} C_VEL
LIN {X 0,Y 509.856,Z 286.971,A -85,B 0,C 180,E1 -5531.425,E2 -5531.425} C_VEL
LIN {X 0,Y 509.839,Z 286.98,A -85,B 0,C 180,E1 -5534.67,E2 -5534.67} C_VEL
LIN {X 0,Y 509.833,Z 286.973,A -85,B 0,C 180,E1 -5537.51,E2 -5537.51} C_VEL
LIN {X 0,Y 509.846,Z 286.977,A -85,B 0,C 180,E1 -5540.647,E2 -5540.647} C_VEL
LIN {X 0,Y 509.824,Z 286.974,A -85,B 0,C 180,E1 -5543.647,E2 -5543.647} C_VEL
LIN {X 0,Y 509.858,Z 286.971,A -85,B 0,C 180,E1 -5546.539,E2 -5546.539} C_VEL
LIN {X 0,Y 509.845,Z 286.975,A -85,B 0,C 180,E1 -5549.334,E2 -5549.334} C_VEL
LIN {X 0,Y 509.891,Z 286.965,A -85,B 0,C 180,E1 -5552.054,E2 -5552.054} C_VEL
LIN {X 0,Y 509.875,Z 286.969,A -85,B 0,C 180,E1 -5554.704,E2 -5554.704} C_VEL
LIN {X 0,Y 509.825,Z 286.98,A -85,B 0,C 180,E1 -5557.458,E2 -5557.458} C_VEL
LIN {X 0,Y 509.915,Z 286.964,A -85,B 0,C 180,E1 -5559.844,E2 -5559.844} C_VEL
LIN {X 0,Y 509.883,Z 286.97,A -85,B 0,C 180,E1 -5563.175,E2 -5563.175} C_VEL
LIN {X 0,Y 509.872,Z 286.973,A -85,B 0,C 180,E1 -5565.634,E2 -5565.634} C_VEL
LIN {X 0,Y 509.911,Z 286.962,A -85,B 0,C 180,E1 -5568.874,E2 -5568.874} C_VEL
LIN {X 0,Y 509.949,Z 286.961,A -85,B 0,C 180,E1 -5572.078,E2 -5572.078} C_VEL
LIN {X 0,Y 509.978,Z 286.952,A -85,B 0,C 180,E1 -5574.464,E2 -5574.464} C_VEL
LIN {X 0,Y 510.053,Z 286.948,A -85,B 0,C 180,E1 -5577.631,E2 -5577.631} C_VEL
LIN {X 0,Y 510.061,Z 286.943,A -85,B 0,C 180,E1 -5580.789,E2 -5580.789} C_VEL
LIN {X 0,Y 509.953,Z 286.954,A -85,B 0,C 180,E1 -5583.16,E2 -5583.16} C_VEL
LIN {X 0,Y 509.952,Z 286.963,A -85,B 0,C 180,E1 -5586.33,E2 -5586.33} C_VEL
LIN {X 0,Y 509.912,Z 286.965,A -85,B 0,C 180,E1 -5588.72,E2 -5588.72} C_VEL
LIN {X 0,Y 509.902,Z 286.965,A -85,B 0,C 180,E1 -5591.932,E2 -5591.932} C_VEL
LIN {X 0,Y 509.892,Z 286.965,A -85,B 0,C 180,E1 -5595.242,E2 -5595.242} C_VEL
LIN {X 0,Y 509.887,Z 286.967,A -85,B 0,C 180,E1 -5598.001,E2 -5598.001} C_VEL
LIN {X 0,Y 509.848,Z 286.974,A -85,B 0,C 180,E1 -5601.002,E2 -5601.002} C_VEL
LIN {X 0,Y 509.868,Z 286.971,A -85,B 0,C 180,E1 -5604.426,E2 -5604.426} C_VEL
LIN {X 0,Y 509.882,Z 286.971,A -85,B 0,C 180,E1 -5607.056,E2 -5607.056} C_VEL
LIN {X 0,Y 509.856,Z 286.969,A -85,B 0,C 180,E1 -5609.751,E2 -5609.751} C_VEL
LIN {X 0,Y 509.871,Z 286.971,A -85,B 0,C 180,E1 -5612.774,E2 -5612.774} C_VEL
LIN {X 0,Y 509.824,Z 286.977,A -85,B 0,C 180,E1 -5615.579,E2 -5615.579} C_VEL
LIN {X 0,Y 509.849,Z 286.97,A -85,B 0,C 180,E1 -5618.338,E2 -5618.338} C_VEL
LIN {X 0,Y 509.855,Z 286.978,A -85,B 0,C 180,E1 -5621.426,E2 -5621.426} C_VEL
LIN {X 0,Y 509.838,Z 286.973,A -85,B 0,C 180,E1 -5624.67,E2 -5624.67} C_VEL
LIN {X 0,Y 509.855,Z 286.972,A -85,B 0,C 180,E1 -5628.104,E2 -5628.104} C_VEL
LIN {X 0,Y 509.845,Z 286.972,A -85,B 0,C 180,E1 -5630.648,E2 -5630.648} C_VEL
LIN {X 0,Y 509.821,Z 286.983,A -85,B 0,C 180,E1 -5633.729,E2 -5633.729} C_VEL
LIN {X 0,Y 509.152,Z 287.06,A -85,B 0,C 180,E1 -5634.388,E2 -5634.388} C_VEL
LIN {X 0,Y 506.341,Z 287.413,A -85,B 0,C 180,E1 -5635.461,E2 -5635.461} C_VEL
LIN {X 0,Y 503.955,Z 287.71,A -85,B 0,C 180,E1 -5636.324,E2 -5636.324} C_VEL
LIN {X 0,Y 502.907,Z 287.839,A -85,B 0,C 180,E1 -5636.99,E2 -5636.99} C_VEL
LIN {X 0,Y 502.809,Z 287.851,A -85,B 0,C 180,E1 -5637.216,E2 -5637.216} C_VEL
LIN {X 0,Y 502.898,Z 288.044,A -85,B 0,C 180,E1 -5640.18,E2 -5640.18} C_VEL
LIN {X 0,Y 503.453,Z 293.401,A -85,B 0,C 180,E1 -5641.21,E2 -5641.21} C_VEL
LIN {X 0,Y 503.268,Z 309.837,A -85,B 0,C 180,E1 -5644.251,E2 -5644.251} C_VEL
LIN {X 0,Y 505.504,Z 322.386,A -85,B 0,C 180,E1 -5644.507,E2 -5644.507} C_VEL
LIN {X 0,Y 504.836,Z 416.345,A -85,B 0,C 180,E1 -5645.862,E2 -5645.862} C_VEL
LIN {X 0,Y 504.638,Z 429.455,A -85,B 0,C 180,E1 -5646.206,E2 -5646.206} C_VEL
LIN {X 0,Y 504.401,Z 442.013,A -85,B 0,C 180,E1 -5646.7,E2 -5646.7} C_VEL
LIN {X 0,Y 504.093,Z 454.127,A -85,B 0,C 180,E1 -5647.347,E2 -5647.347} C_VEL
LIN {X 0,Y 503.736,Z 464.824,A -85,B 0,C 180,E1 -5648.086,E2 -5648.086} C_VEL
LIN {X 0,Y 503.425,Z 474.352,A -85,B 0,C 180,E1 -5648.899,E2 -5648.899} C_VEL
LIN {X 0,Y 503.065,Z 484.688,A -85,B 0,C 180,E1 -5649.984,E2 -5649.984} C_VEL
LIN {X 0,Y 502.827,Z 492.794,A -85,B 0,C 180,E1 -5651.036,E2 -5651.036} C_VEL
LIN {X 0,Y 502.53,Z 500.601,A -85,B 0,C 180,E1 -5652.291,E2 -5652.291} C_VEL
LIN {X 0,Y 502.362,Z 505.887,A -85,B 0,C 180,E1 -5653.334,E2 -5653.334} C_VEL
LIN {X 0,Y 502.246,Z 510.954,A -85,B 0,C 180,E1 -5654.581,E2 -5654.581} C_VEL
LIN {X 0,Y 502.162,Z 514.824,A -85,B 0,C 180,E1 -5655.823,E2 -5655.823} C_VEL
LIN {X 0,Y 502.06,Z 517.615,A -85,B 0,C 180,E1 -5657.057,E2 -5657.057} C_VEL
LIN {X 0,Y 502.104,Z 519.582,A -85,B 0,C 180,E1 -5658.463,E2 -5658.463} C_VEL
LIN {X 0,Y 502.064,Z 520.272,A -85,B 0,C 180,E1 -5659.515,E2 -5659.515} C_VEL
LIN {X 0,Y 502.039,Z 519.979,A -85,B 0,C 180,E1 -5661.142,E2 -5661.142} C_VEL
LIN {X 0,Y 502.091,Z 519.249,A -85,B 0,C 180,E1 -5661.953,E2 -5661.953} C_VEL
LIN {X 0,Y 502.194,Z 516.604,A -85,B 0,C 180,E1 -5663.523,E2 -5663.523} C_VEL
LIN {X 0,Y 502.176,Z 513.34,A -85,B 0,C 180,E1 -5664.78,E2 -5664.78} C_VEL
LIN {X 0,Y 502.279,Z 509.128,A -85,B 0,C 180,E1 -5665.988,E2 -5665.988} C_VEL
LIN {X 0,Y 502.45,Z 502.761,A -85,B 0,C 180,E1 -5667.394,E2 -5667.394} C_VEL
LIN {X 0,Y 502.65,Z 495.816,A -85,B 0,C 180,E1 -5668.598,E2 -5668.598} C_VEL
LIN {X 0,Y 502.975,Z 487.15,A -85,B 0,C 180,E1 -5669.799,E2 -5669.799} C_VEL
LIN {X 0,Y 503.21,Z 478.321,A -85,B 0,C 180,E1 -5670.8,E2 -5670.8} C_VEL
LIN {X 0,Y 503.513,Z 468.627,A -85,B 0,C 180,E1 -5671.699,E2 -5671.699} C_VEL
LIN {X 0,Y 503.981,Z 457.898,A -85,B 0,C 180,E1 -5672.497,E2 -5672.497} C_VEL
LIN {X 0,Y 504.321,Z 445.953,A -85,B 0,C 180,E1 -5673.195,E2 -5673.195} C_VEL
LIN {X 0,Y 504.608,Z 433.491,A -85,B 0,C 180,E1 -5673.743,E2 -5673.743} C_VEL
LIN {X 0,Y 504.832,Z 422.281,A -85,B 0,C 180,E1 -5674.091,E2 -5674.091} C_VEL
LIN {X 0,Y 504.948,Z 409.409,A -85,B 0,C 180,E1 -5674.34,E2 -5674.34} C_VEL
LIN {X 0,Y 505.336,Z 321.01,A -85,B 0,C 180,E1 -5675.606,E2 -5675.606} C_VEL
LIN {X 0,Y 503.204,Z 309.676,A -85,B 0,C 180,E1 -5675.861,E2 -5675.861} C_VEL
LIN {X 0,Y 503.458,Z 296.201,A -85,B 0,C 180,E1 -5678.428,E2 -5678.428} C_VEL
LIN {X 0,Y 503.364,Z 290.956,A -85,B 0,C 180,E1 -5679.442,E2 -5679.442} C_VEL
LIN {X 0,Y 502.798,Z 287.858,A -85,B 0,C 180,E1 -5680.062,E2 -5680.062} C_VEL
LIN {X 0,Y 502.842,Z 287.852,A -85,B 0,C 180,E1 -5682.101,E2 -5682.101} C_VEL
LIN {X 0,Y 502.847,Z 287.842,A -85,B 0,C 180,E1 -5685.399,E2 -5685.399} C_VEL
LIN {X 0,Y 502.801,Z 287.852,A -85,B 0,C 180,E1 -5688.752,E2 -5688.752} C_VEL
LIN {X 0,Y 502.778,Z 287.851,A -85,B 0,C 180,E1 -5691.311,E2 -5691.311} C_VEL
LIN {X 0,Y 502.763,Z 287.854,A -85,B 0,C 180,E1 -5693.914,E2 -5693.914} C_VEL
LIN {X 0,Y 502.778,Z 287.86,A -85,B 0,C 180,E1 -5696.57,E2 -5696.57} C_VEL
LIN {X 0,Y 502.805,Z 287.848,A -85,B 0,C 180,E1 -5699.933,E2 -5699.933} C_VEL
LIN {X 0,Y 502.825,Z 287.851,A -85,B 0,C 180,E1 -5703.031,E2 -5703.031} C_VEL
LIN {X 0,Y 502.768,Z 287.852,A -85,B 0,C 180,E1 -5705.95,E2 -5705.95} C_VEL
LIN {X 0,Y 502.788,Z 287.859,A -85,B 0,C 180,E1 -5708.976,E2 -5708.976} C_VEL
LIN {X 0,Y 502.765,Z 287.853,A -85,B 0,C 180,E1 -5712.194,E2 -5712.194} C_VEL
LIN {X 0,Y 502.779,Z 287.855,A -85,B 0,C 180,E1 -5715.469,E2 -5715.469} C_VEL
LIN {X 0,Y 502.788,Z 287.851,A -85,B 0,C 180,E1 -5717.86,E2 -5717.86} C_VEL
LIN {X 0,Y 502.787,Z 287.855,A -85,B 0,C 180,E1 -5721.023,E2 -5721.023} C_VEL
LIN {X 0,Y 502.767,Z 287.853,A -85,B 0,C 180,E1 -5724.168,E2 -5724.168} C_VEL
LIN {X 0,Y 502.825,Z 287.848,A -85,B 0,C 180,E1 -5726.993,E2 -5726.993} C_VEL
LIN {X 0,Y 502.807,Z 287.849,A -85,B 0,C 180,E1 -5730.064,E2 -5730.064} C_VEL
LIN {X 0,Y 502.813,Z 287.847,A -85,B 0,C 180,E1 -5732.532,E2 -5732.532} C_VEL
LIN {X 0,Y 502.794,Z 287.853,A -85,B 0,C 180,E1 -5735.305,E2 -5735.305} C_VEL
LIN {X 0,Y 502.771,Z 287.86,A -85,B 0,C 180,E1 -5737.826,E2 -5737.826} C_VEL
LIN {X 0,Y 502.815,Z 287.848,A -85,B 0,C 180,E1 -5740.4,E2 -5740.4} C_VEL
LIN {X 0,Y 502.824,Z 287.845,A -85,B 0,C 180,E1 -5742.931,E2 -5742.931} C_VEL
LIN {X 0,Y 502.834,Z 287.846,A -85,B 0,C 180,E1 -5745.429,E2 -5745.429} C_VEL
LIN {X 0,Y 502.868,Z 287.841,A -85,B 0,C 180,E1 -5748.717,E2 -5748.717} C_VEL
LIN {X 0,Y 502.892,Z 287.844,A -85,B 0,C 180,E1 -5751.967,E2 -5751.967} C_VEL
LIN {X 0,Y 502.919,Z 287.839,A -85,B 0,C 180,E1 -5754.386,E2 -5754.386} C_VEL
LIN {X 0,Y 503.014,Z 287.823,A -85,B 0,C 180,E1 -5757.598,E2 -5757.598} C_VEL
LIN {X 0,Y 503.016,Z 287.826,A -85,B 0,C 180,E1 -5760,E2 -5760} C_VEL
LIN {X 0,Y 503.014,Z 287.831,A -85,B 0,C 180,E1 -5762.402,E2 -5762.402} C_VEL
LIN {X 0,Y 502.929,Z 287.832,A -85,B 0,C 180,E1 -5765.614,E2 -5765.614} C_VEL
LIN {X 0,Y 502.894,Z 287.839,A -85,B 0,C 180,E1 -5768.034,E2 -5768.034} C_VEL
LIN {X 0,Y 502.873,Z 287.84,A -85,B 0,C 180,E1 -5771.283,E2 -5771.283} C_VEL
LIN {X 0,Y 502.843,Z 287.85,A -85,B 0,C 180,E1 -5774.571,E2 -5774.571} C_VEL
LIN {X 0,Y 502.854,Z 287.842,A -85,B 0,C 180,E1 -5777.907,E2 -5777.907} C_VEL
LIN {X 0,Y 502.821,Z 287.85,A -85,B 0,C 180,E1 -5780.537,E2 -5780.537} C_VEL
LIN {X 0,Y 502.787,Z 287.858,A -85,B 0,C 180,E1 -5783.041,E2 -5783.041} C_VEL
LIN {X 0,Y 502.834,Z 287.845,A -85,B 0,C 180,E1 -5785.676,E2 -5785.676} C_VEL
LIN {X 0,Y 502.834,Z 287.845,A -85,B 0,C 180,E1 -5788.373,E2 -5788.373} C_VEL
LIN {X 0,Y 502.791,Z 287.854,A -85,B 0,C 180,E1 -5791.5,E2 -5791.5} C_VEL
LIN {X 0,Y 502.798,Z 287.849,A -85,B 0,C 180,E1 -5794.445,E2 -5794.445} C_VEL
LIN {X 0,Y 502.777,Z 287.859,A -85,B 0,C 180,E1 -5797.179,E2 -5797.179} C_VEL
LIN {X 0,Y 502.783,Z 287.852,A -85,B 0,C 180,E1 -5800.016,E2 -5800.016} C_VEL
LIN {X 0,Y 502.798,Z 287.849,A -85,B 0,C 180,E1 -5802.2,E2 -5802.2} C_VEL
LIN {X 0,Y 502.797,Z 287.857,A -85,B 0,C 180,E1 -5805.469,E2 -5805.469} C_VEL
LIN {X 0,Y 502.817,Z 287.847,A -85,B 0,C 180,E1 -5808.935,E2 -5808.935} C_VEL
LIN {X 0,Y 502.79,Z 287.854,A -85,B 0,C 180,E1 -5812.047,E2 -5812.047} C_VEL
LIN {X 0,Y 502.797,Z 287.849,A -85,B 0,C 180,E1 -5815.035,E2 -5815.035} C_VEL
LIN {X 0,Y 502.781,Z 287.859,A -85,B 0,C 180,E1 -5817.916,E2 -5817.916} C_VEL
LIN {X 0,Y 502.823,Z 287.848,A -85,B 0,C 180,E1 -5820.713,E2 -5820.713} C_VEL
LIN {X 0,Y 502.862,Z 287.845,A -85,B 0,C 180,E1 -5823.44,E2 -5823.44} C_VEL
LIN {X 0,Y 502.875,Z 288.014,A -85,B 0,C 180,E1 -5824.953,E2 -5824.953} C_VEL
LIN {X 0,Y 504.548,Z 297.278,A -85,B 0,C 180,E1 -5826.555,E2 -5826.555} C_VEL
LIN {X 0,Y 504.101,Z 314.474,A -85,B 0,C 180,E1 -5829.342,E2 -5829.342} C_VEL
LIN {X 0,Y 503.547,Z 333.152,A -85,B 0,C 180,E1 -5832.329,E2 -5832.329} C_VEL
LIN {X 0,Y 503.256,Z 344.879,A -85,B 0,C 180,E1 -5834.19,E2 -5834.19} C_VEL
LIN {X 0,Y 505.322,Z 359.991,A -85,B 0,C 180,E1 -5834.476,E2 -5834.476} C_VEL
LIN {X 0,Y 504.831,Z 453.132,A -85,B 0,C 180,E1 -5835.823,E2 -5835.823} C_VEL
LIN {X 0,Y 504.536,Z 466.462,A -85,B 0,C 180,E1 -5836.174,E2 -5836.174} C_VEL
LIN {X 0,Y 504.244,Z 478.662,A -85,B 0,C 180,E1 -5836.654,E2 -5836.654} C_VEL
LIN {X 0,Y 503.948,Z 490.627,A -85,B 0,C 180,E1 -5837.29,E2 -5837.29} C_VEL
LIN {X 0,Y 503.527,Z 502.596,A -85,B 0,C 180,E1 -5838.12,E2 -5838.12} C_VEL
LIN {X 0,Y 503.217,Z 513.063,A -85,B 0,C 180,E1 -5839.031,E2 -5839.031} C_VEL
LIN {X 0,Y 502.872,Z 521.62,A -85,B 0,C 180,E1 -5839.94,E2 -5839.94} C_VEL
LIN {X 0,Y 502.628,Z 529.518,A -85,B 0,C 180,E1 -5840.95,E2 -5840.95} C_VEL
LIN {X 0,Y 502.399,Z 537.232,A -85,B 0,C 180,E1 -5842.161,E2 -5842.161} C_VEL
LIN {X 0,Y 502.235,Z 544.343,A -85,B 0,C 180,E1 -5843.573,E2 -5843.573} C_VEL
LIN {X 0,Y 502.174,Z 549.076,A -85,B 0,C 180,E1 -5844.781,E2 -5844.781} C_VEL
LIN {X 0,Y 502.139,Z 552.691,A -85,B 0,C 180,E1 -5845.988,E2 -5845.988} C_VEL
LIN {X 0,Y 502.12,Z 554.556,A -85,B 0,C 180,E1 -5846.791,E2 -5846.791} C_VEL
LIN {X 0,Y 502.091,Z 555.953,A -85,B 0,C 180,E1 -5847.594,E2 -5847.594} C_VEL
LIN {X 0,Y 501.99,Z 557.554,A -85,B 0,C 180,E1 -5849.198,E2 -5849.198} C_VEL
LIN {X 0,Y 501.983,Z 557.769,A -85,B 0,C 180,E1 -5850,E2 -5850} C_VEL
LIN {X 0,Y 502.036,Z 556.943,A -85,B 0,C 180,E1 -5851.605,E2 -5851.605} C_VEL
LIN {X 0,Y 502.091,Z 555.945,A -85,B 0,C 180,E1 -5852.407,E2 -5852.407} C_VEL
LIN {X 0,Y 502.12,Z 554.546,A -85,B 0,C 180,E1 -5853.21,E2 -5853.21} C_VEL
LIN {X 0,Y 502.102,Z 551.599,A -85,B 0,C 180,E1 -5854.416,E2 -5854.416} C_VEL
LIN {X 0,Y 502.21,Z 547.616,A -85,B 0,C 180,E1 -5855.622,E2 -5855.622} C_VEL
LIN {X 0,Y 502.331,Z 541.59,A -85,B 0,C 180,E1 -5857.012,E2 -5857.012} C_VEL
LIN {X 0,Y 502.477,Z 534.792,A -85,B 0,C 180,E1 -5858.243,E2 -5858.243} C_VEL
LIN {X 0,Y 502.713,Z 526.487,A -85,B 0,C 180,E1 -5859.455,E2 -5859.455} C_VEL
LIN {X 0,Y 502.989,Z 517.976,A -85,B 0,C 180,E1 -5860.466,E2 -5860.466} C_VEL
LIN {X 0,Y 503.416,Z 507.464,A -85,B 0,C 180,E1 -5861.475,E2 -5861.475} C_VEL
LIN {X 0,Y 503.738,Z 495.993,A -85,B 0,C 180,E1 -5862.361,E2 -5862.361} C_VEL
LIN {X 0,Y 504.059,Z 485.662,A -85,B 0,C 180,E1 -5862.993,E2 -5862.993} C_VEL
LIN {X 0,Y 504.372,Z 473.954,A -85,B 0,C 180,E1 -5863.549,E2 -5863.549} C_VEL
LIN {X 0,Y 504.686,Z 460.468,A -85,B 0,C 180,E1 -5864.002,E2 -5864.002} C_VEL
LIN {X 0,Y 504.889,Z 447.08,A -85,B 0,C 180,E1 -5864.279,E2 -5864.279} C_VEL
LIN {X 0,Y 505.255,Z 357.908,A -85,B 0,C 180,E1 -5865.555,E2 -5865.555} C_VEL
LIN {X 0,Y 503.227,Z 344.738,A -85,B 0,C 180,E1 -5865.82,E2 -5865.82} C_VEL
LIN {X 0,Y 503.764,Z 325.145,A -85,B 0,C 180,E1 -5868.927,E2 -5868.927} C_VEL
LIN {X 0,Y 504.285,Z 306.757,A -85,B 0,C 180,E1 -5871.889,E2 -5871.889} C_VEL
LIN {X 0,Y 504.553,Z 297.254,A -85,B 0,C 180,E1 -5873.442,E2 -5873.442} C_VEL
LIN {X 0,Y 502.867,Z 287.846,A -85,B 0,C 180,E1 -5875.109,E2 -5875.109} C_VEL
LIN {X 0,Y 502.832,Z 287.852,A -85,B 0,C 180,E1 -5877.467,E2 -5877.467} C_VEL
LIN {X 0,Y 502.812,Z 287.856,A -85,B 0,C 180,E1 -5880.211,E2 -5880.211} C_VEL
LIN {X 0,Y 502.834,Z 287.845,A -85,B 0,C 180,E1 -5883.031,E2 -5883.031} C_VEL
LIN {X 0,Y 502.775,Z 287.857,A -85,B 0,C 180,E1 -5885.951,E2 -5885.951} C_VEL
LIN {X 0,Y 502.802,Z 287.851,A -85,B 0,C 180,E1 -5888.976,E2 -5888.976} C_VEL
LIN {X 0,Y 502.796,Z 287.854,A -85,B 0,C 180,E1 -5892.139,E2 -5892.139} C_VEL
LIN {X 0,Y 502.786,Z 287.851,A -85,B 0,C 180,E1 -5895.47,E2 -5895.47} C_VEL
LIN {X 0,Y 502.82,Z 287.851,A -85,B 0,C 180,E1 -5898.934,E2 -5898.934} C_VEL
LIN {X 0,Y 502.793,Z 287.85,A -85,B 0,C 180,E1 -5902.046,E2 -5902.046} C_VEL
LIN {X 0,Y 502.798,Z 287.854,A -85,B 0,C 180,E1 -5905.034,E2 -5905.034} C_VEL
LIN {X 0,Y 502.782,Z 287.851,A -85,B 0,C 180,E1 -5907.915,E2 -5907.915} C_VEL
LIN {X 0,Y 502.823,Z 287.848,A -85,B 0,C 180,E1 -5910.712,E2 -5910.712} C_VEL
LIN {X 0,Y 502.862,Z 287.846,A -85,B 0,C 180,E1 -5913.439,E2 -5913.439} C_VEL
LIN {X 0,Y 502.784,Z 287.85,A -85,B 0,C 180,E1 -5916.086,E2 -5916.086} C_VEL
LIN {X 0,Y 502.782,Z 287.851,A -85,B 0,C 180,E1 -5918.689,E2 -5918.689} C_VEL
LIN {X 0,Y 502.829,Z 287.851,A -85,B 0,C 180,E1 -5921.248,E2 -5921.248} C_VEL
LIN {X 0,Y 502.821,Z 287.85,A -85,B 0,C 180,E1 -5923.767,E2 -5923.767} C_VEL
LIN {X 0,Y 502.833,Z 287.844,A -85,B 0,C 180,E1 -5926.255,E2 -5926.255} C_VEL
LIN {X 0,Y 502.875,Z 287.838,A -85,B 0,C 180,E1 -5928.717,E2 -5928.717} C_VEL
LIN {X 0,Y 502.9,Z 287.841,A -85,B 0,C 180,E1 -5931.967,E2 -5931.967} C_VEL
LIN {X 0,Y 502.935,Z 287.83,A -85,B 0,C 180,E1 -5934.386,E2 -5934.386} C_VEL
LIN {X 0,Y 503.023,Z 287.824,A -85,B 0,C 180,E1 -5937.598,E2 -5937.598} C_VEL
LIN {X 0,Y 503.025,Z 287.825,A -85,B 0,C 180,E1 -5940,E2 -5940} C_VEL
LIN {X 0,Y 503.022,Z 287.822,A -85,B 0,C 180,E1 -5942.402,E2 -5942.402} C_VEL
LIN {X 0,Y 502.93,Z 287.833,A -85,B 0,C 180,E1 -5945.613,E2 -5945.613} C_VEL
LIN {X 0,Y 502.899,Z 287.839,A -85,B 0,C 180,E1 -5948.033,E2 -5948.033} C_VEL
LIN {X 0,Y 502.875,Z 287.838,A -85,B 0,C 180,E1 -5951.283,E2 -5951.283} C_VEL
LIN {X 0,Y 502.85,Z 287.85,A -85,B 0,C 180,E1 -5954.571,E2 -5954.571} C_VEL
LIN {X 0,Y 502.86,Z 287.842,A -85,B 0,C 180,E1 -5957.907,E2 -5957.907} C_VEL
LIN {X 0,Y 502.827,Z 287.852,A -85,B 0,C 180,E1 -5960.536,E2 -5960.536} C_VEL
LIN {X 0,Y 502.793,Z 287.854,A -85,B 0,C 180,E1 -5963.04,E2 -5963.04} C_VEL
LIN {X 0,Y 502.839,Z 287.843,A -85,B 0,C 180,E1 -5965.676,E2 -5965.676} C_VEL
LIN {X 0,Y 502.838,Z 287.844,A -85,B 0,C 180,E1 -5968.373,E2 -5968.373} C_VEL
LIN {X 0,Y 502.791,Z 287.85,A -85,B 0,C 180,E1 -5971.499,E2 -5971.499} C_VEL
LIN {X 0,Y 502.802,Z 287.847,A -85,B 0,C 180,E1 -5973.994,E2 -5973.994} C_VEL
LIN {X 0,Y 502.776,Z 287.859,A -85,B 0,C 180,E1 -5977.178,E2 -5977.178} C_VEL
LIN {X 0,Y 502.787,Z 287.85,A -85,B 0,C 180,E1 -5980.015,E2 -5980.015} C_VEL
LIN {X 0,Y 502.802,Z 287.849,A -85,B 0,C 180,E1 -5982.199,E2 -5982.199} C_VEL
LIN {X 0,Y 502.785,Z 287.859,A -85,B 0,C 180,E1 -5985.47,E2 -5985.47} C_VEL
LIN {X 0,Y 502.819,Z 287.848,A -85,B 0,C 180,E1 -5988.934,E2 -5988.934} C_VEL
LIN {X 0,Y 502.793,Z 287.853,A -85,B 0,C 180,E1 -5992.046,E2 -5992.046} C_VEL
LIN {X 0,Y 502.799,Z 287.85,A -85,B 0,C 180,E1 -5995.034,E2 -5995.034} C_VEL
LIN {X 0,Y 502.809,Z 287.851,A -85,B 0,C 180,E1 -5997.216,E2 -5997.216} C_VEL
LIN {X 0,Y 502.107,Z 287.944,A -85,B 0,C 180,E1 -5997.662,E2 -5997.662} C_VEL
LIN {X 0,Y 496.422,Z 288.65,A -85,B 0,C 180,E1 -5999.065,E2 -5999.065} C_VEL
LIN {X 0,Y 495.768,Z 288.733,A -85,B 0,C 180,E1 -5999.52,E2 -5999.52} C_VEL
LIN {X 0,Y 495.81,Z 288.798,A -85,B 0,C 180,E1 -5999.998,E2 -5999.998} C_VEL
LIN {X 0,Y 496.491,Z 293.905,A -85,B 0,C 180,E1 -6000.999,E2 -6000.999} C_VEL
LIN {X 0,Y 496.274,Z 309.916,A -85,B 0,C 180,E1 -6004.008,E2 -6004.008} C_VEL
LIN {X 0,Y 498.659,Z 322.448,A -85,B 0,C 180,E1 -6004.281,E2 -6004.281} C_VEL
LIN {X 0,Y 497.972,Z 417.273,A -85,B 0,C 180,E1 -6005.674,E2 -6005.674} C_VEL
LIN {X 0,Y 497.717,Z 430.931,A -85,B 0,C 180,E1 -6006.049,E2 -6006.049} C_VEL
LIN {X 0,Y 497.498,Z 443.182,A -85,B 0,C 180,E1 -6006.551,E2 -6006.551} C_VEL
LIN {X 0,Y 497.165,Z 455.414,A -85,B 0,C 180,E1 -6007.233,E2 -6007.233} C_VEL
LIN {X 0,Y 496.694,Z 467.247,A -85,B 0,C 180,E1 -6008.087,E2 -6008.087} C_VEL
LIN {X 0,Y 496.349,Z 478.011,A -85,B 0,C 180,E1 -6009.074,E2 -6009.074} C_VEL
LIN {X 0,Y 495.971,Z 487.195,A -85,B 0,C 180,E1 -6010.118,E2 -6010.118} C_VEL
LIN {X 0,Y 495.691,Z 496.278,A -85,B 0,C 180,E1 -6011.397,E2 -6011.397} C_VEL
LIN {X 0,Y 495.465,Z 503.435,A -85,B 0,C 180,E1 -6012.67,E2 -6012.67} C_VEL
LIN {X 0,Y 495.257,Z 509.094,A -85,B 0,C 180,E1 -6013.935,E2 -6013.935} C_VEL
LIN {X 0,Y 495.14,Z 513.487,A -85,B 0,C 180,E1 -6015.197,E2 -6015.197} C_VEL
LIN {X 0,Y 495.072,Z 515.795,A -85,B 0,C 180,E1 -6016.035,E2 -6016.035} C_VEL
LIN {X 0,Y 494.988,Z 517.623,A -85,B 0,C 180,E1 -6016.869,E2 -6016.869} C_VEL
LIN {X 0,Y 495.007,Z 519.828,A -85,B 0,C 180,E1 -6018.42,E2 -6018.42} C_VEL
LIN {X 0,Y 494.973,Z 520.496,A -85,B 0,C 180,E1 -6019.363,E2 -6019.363} C_VEL
LIN {X 0,Y 494.935,Z 520.612,A -85,B 0,C 180,E1 -6020.189,E2 -6020.189} C_VEL
LIN {X 0,Y 494.992,Z 519.654,A -85,B 0,C 180,E1 -6021.837,E2 -6021.837} C_VEL
LIN {X 0,Y 495.013,Z 518.59,A -85,B 0,C 180,E1 -6022.658,E2 -6022.658} C_VEL
LIN {X 0,Y 495.11,Z 516.951,A -85,B 0,C 180,E1 -6023.534,E2 -6023.534} C_VEL
LIN {X 0,Y 495.111,Z 514.031,A -85,B 0,C 180,E1 -6024.706,E2 -6024.706} C_VEL
LIN {X 0,Y 495.209,Z 509.948,A -85,B 0,C 180,E1 -6025.931,E2 -6025.931} C_VEL
LIN {X 0,Y 495.38,Z 503.718,A -85,B 0,C 180,E1 -6027.357,E2 -6027.357} C_VEL
LIN {X 0,Y 495.574,Z 496.959,A -85,B 0,C 180,E1 -6028.577,E2 -6028.577} C_VEL
LIN {X 0,Y 495.919,Z 488.531,A -85,B 0,C 180,E1 -6029.797,E2 -6029.797} C_VEL
LIN {X 0,Y 496.189,Z 479.915,A -85,B 0,C 180,E1 -6030.811,E2 -6030.811} C_VEL
LIN {X 0,Y 496.534,Z 469.334,A -85,B 0,C 180,E1 -6031.825,E2 -6031.825} C_VEL
LIN {X 0,Y 497.033,Z 458.743,A -85,B 0,C 180,E1 -6032.633,E2 -6032.633} C_VEL
LIN {X 0,Y 497.389,Z 446.951,A -85,B 0,C 180,E1 -6033.341,E2 -6033.341} C_VEL
LIN {X 0,Y 497.702,Z 434.705,A -85,B 0,C 180,E1 -6033.896,E2 -6033.896} C_VEL
LIN {X 0,Y 497.899,Z 423.907,A -85,B 0,C 180,E1 -6034.249,E2 -6034.249} C_VEL
LIN {X 0,Y 498.074,Z 410.526,A -85,B 0,C 180,E1 -6034.527,E2 -6034.527} C_VEL
LIN {X 0,Y 498.59,Z 322.45,A -85,B 0,C 180,E1 -6035.802,E2 -6035.802} C_VEL
LIN {X 0,Y 496.235,Z 309.956,A -85,B 0,C 180,E1 -6036.071,E2 -6036.071} C_VEL
LIN {X 0,Y 496.476,Z 295.977,A -85,B 0,C 180,E1 -6038.752,E2 -6038.752} C_VEL
LIN {X 0,Y 496.324,Z 291.746,A -85,B 0,C 180,E1 -6039.577,E2 -6039.577} C_VEL
LIN {X 0,Y 495.754,Z 288.736,A -85,B 0,C 180,E1 -6040.206,E2 -6040.206} C_VEL
LIN {X 0,Y 495.784,Z 288.732,A -85,B 0,C 180,E1 -6042.276,E2 -6042.276} C_VEL
LIN {X 0,Y 495.804,Z 288.721,A -85,B 0,C 180,E1 -6045.623,E2 -6045.623} C_VEL
LIN {X 0,Y 495.761,Z 288.727,A -85,B 0,C 180,E1 -6049.029,E2 -6049.029} C_VEL
LIN {X 0,Y 495.738,Z 288.728,A -85,B 0,C 180,E1 -6051.628,E2 -6051.628} C_VEL
LIN {X 0,Y 495.709,Z 288.737,A -85,B 0,C 180,E1 -6054.276,E2 -6054.276} C_VEL
LIN {X 0,Y 495.726,Z 288.734,A -85,B 0,C 180,E1 -6056.978,E2 -6056.978} C_VEL
LIN {X 0,Y 495.753,Z 288.728,A -85,B 0,C 180,E1 -6060.144,E2 -6060.144} C_VEL
LIN {X 0,Y 495.785,Z 288.725,A -85,B 0,C 180,E1 -6063.243,E2 -6063.243} C_VEL
LIN {X 0,Y 495.715,Z 288.731,A -85,B 0,C 180,E1 -6066.088,E2 -6066.088} C_VEL
LIN {X 0,Y 495.753,Z 288.733,A -85,B 0,C 180,E1 -6068.767,E2 -6068.767} C_VEL
LIN {X 0,Y 495.737,Z 288.729,A -85,B 0,C 180,E1 -6071.782,E2 -6071.782} C_VEL
LIN {X 0,Y 495.731,Z 288.738,A -85,B 0,C 180,E1 -6075.14,E2 -6075.14} C_VEL
LIN {X 0,Y 495.744,Z 288.727,A -85,B 0,C 180,E1 -6078.218,E2 -6078.218} C_VEL
LIN {X 0,Y 495.739,Z 288.735,A -85,B 0,C 180,E1 -6081.407,E2 -6081.407} C_VEL
LIN {X 0,Y 495.74,Z 288.728,A -85,B 0,C 180,E1 -6084.462,E2 -6084.462} C_VEL
LIN {X 0,Y 495.759,Z 288.734,A -85,B 0,C 180,E1 -6087.405,E2 -6087.405} C_VEL
LIN {X 0,Y 495.757,Z 288.726,A -85,B 0,C 180,E1 -6090.253,E2 -6090.253} C_VEL
LIN {X 0,Y 495.803,Z 288.724,A -85,B 0,C 180,E1 -6093.253,E2 -6093.253} C_VEL
LIN {X 0,Y 495.734,Z 288.728,A -85,B 0,C 180,E1 -6096.612,E2 -6096.612} C_VEL
LIN {X 0,Y 495.769,Z 288.727,A -85,B 0,C 180,E1 -6099.324,E2 -6099.324} C_VEL
LIN {X 0,Y 495.789,Z 288.731,A -85,B 0,C 180,E1 -6101.829,E2 -6101.829} C_VEL
LIN {X 0,Y 495.815,Z 288.72,A -85,B 0,C 180,E1 -6104.548,E2 -6104.548} C_VEL
LIN {X 0,Y 495.819,Z 288.727,A -85,B 0,C 180,E1 -6107.965,E2 -6107.965} C_VEL
LIN {X 0,Y 495.833,Z 288.716,A -85,B 0,C 180,E1 -6111.03,E2 -6111.03} C_VEL
LIN {X 0,Y 495.874,Z 288.718,A -85,B 0,C 180,E1 -6114.306,E2 -6114.306} C_VEL
LIN {X 0,Y 495.983,Z 288.698,A -85,B 0,C 180,E1 -6117.564,E2 -6117.564} C_VEL
LIN {X 0,Y 495.996,Z 288.698,A -85,B 0,C 180,E1 -6120.812,E2 -6120.812} C_VEL
LIN {X 0,Y 495.835,Z 288.716,A -85,B 0,C 180,E1 -6123.25,E2 -6123.25} C_VEL
LIN {X 0,Y 495.87,Z 288.721,A -85,B 0,C 180,E1 -6126.511,E2 -6126.511} C_VEL
LIN {X 0,Y 495.837,Z 288.719,A -85,B 0,C 180,E1 -6128.97,E2 -6128.97} C_VEL
LIN {X 0,Y 495.821,Z 288.719,A -85,B 0,C 180,E1 -6132.036,E2 -6132.036} C_VEL
LIN {X 0,Y 495.815,Z 288.719,A -85,B 0,C 180,E1 -6135.452,E2 -6135.452} C_VEL
LIN {X 0,Y 495.799,Z 288.722,A -85,B 0,C 180,E1 -6138.248,E2 -6138.248} C_VEL
LIN {X 0,Y 495.766,Z 288.732,A -85,B 0,C 180,E1 -6140.757,E2 -6140.757} C_VEL
LIN {X 0,Y 495.744,Z 288.73,A -85,B 0,C 180,E1 -6143.388,E2 -6143.388} C_VEL
LIN {X 0,Y 495.792,Z 288.721,A -85,B 0,C 180,E1 -6146.068,E2 -6146.068} C_VEL
LIN {X 0,Y 495.772,Z 288.729,A -85,B 0,C 180,E1 -6148.815,E2 -6148.815} C_VEL
LIN {X 0,Y 495.753,Z 288.728,A -85,B 0,C 180,E1 -6151.727,E2 -6151.727} C_VEL
LIN {X 0,Y 495.768,Z 288.726,A -85,B 0,C 180,E1 -6154.696,E2 -6154.696} C_VEL
LIN {X 0,Y 495.728,Z 288.735,A -85,B 0,C 180,E1 -6157.562,E2 -6157.562} C_VEL
LIN {X 0,Y 495.762,Z 288.726,A -85,B 0,C 180,E1 -6160.701,E2 -6160.701} C_VEL
LIN {X 0,Y 495.73,Z 288.735,A -85,B 0,C 180,E1 -6163.696,E2 -6163.696} C_VEL
LIN {X 0,Y 495.725,Z 288.73,A -85,B 0,C 180,E1 -6166.306,E2 -6166.306} C_VEL
LIN {X 0,Y 495.763,Z 288.729,A -85,B 0,C 180,E1 -6169.301,E2 -6169.301} C_VEL
LIN {X 0,Y 495.726,Z 288.73,A -85,B 0,C 180,E1 -6172.439,E2 -6172.439} C_VEL
LIN {X 0,Y 495.776,Z 288.728,A -85,B 0,C 180,E1 -6175.458,E2 -6175.458} C_VEL
LIN {X 0,Y 495.754,Z 288.729,A -85,B 0,C 180,E1 -6178.365,E2 -6178.365} C_VEL
LIN {X 0,Y 495.787,Z 288.728,A -85,B 0,C 180,E1 -6181.508,E2 -6181.508} C_VEL
LIN {X 0,Y 495.824,Z 288.725,A -85,B 0,C 180,E1 -6184.611,E2 -6184.611} C_VEL
LIN {X 0,Y 495.83,Z 288.854,A -85,B 0,C 180,E1 -6184.78,E2 -6184.78} C_VEL
LIN {X 0,Y 497.615,Z 298.718,A -85,B 0,C 180,E1 -6186.508,E2 -6186.508} C_VEL
LIN {X 0,Y 497.067,Z 317.075,A -85,B 0,C 180,E1 -6189.517,E2 -6189.517} C_VEL
LIN {X 0,Y 496.493,Z 335.48,A -85,B 0,C 180,E1 -6192.495,E2 -6192.495} C_VEL
LIN {X 0,Y 496.252,Z 344.624,A -85,B 0,C 180,E1 -6193.965,E2 -6193.965} C_VEL
LIN {X 0,Y 498.488,Z 360.658,A -85,B 0,C 180,E1 -6194.274,E2 -6194.274} C_VEL
LIN {X 0,Y 497.94,Z 452.813,A -85,B 0,C 180,E1 -6195.622,E2 -6195.622} C_VEL
LIN {X 0,Y 497.648,Z 466.169,A -85,B 0,C 180,E1 -6195.979,E2 -6195.979} C_VEL
LIN {X 0,Y 497.32,Z 478.382,A -85,B 0,C 180,E1 -6196.465,E2 -6196.465} C_VEL
LIN {X 0,Y 496.994,Z 490.653,A -85,B 0,C 180,E1 -6197.128,E2 -6197.128} C_VEL
LIN {X 0,Y 496.522,Z 502.325,A -85,B 0,C 180,E1 -6197.95,E2 -6197.95} C_VEL
LIN {X 0,Y 496.195,Z 512.794,A -85,B 0,C 180,E1 -6198.874,E2 -6198.874} C_VEL
LIN {X 0,Y 495.847,Z 521.352,A -85,B 0,C 180,E1 -6199.796,E2 -6199.796} C_VEL
LIN {X 0,Y 495.571,Z 529.251,A -85,B 0,C 180,E1 -6200.82,E2 -6200.82} C_VEL
LIN {X 0,Y 495.341,Z 536.967,A -85,B 0,C 180,E1 -6202.049,E2 -6202.049} C_VEL
LIN {X 0,Y 495.164,Z 544.079,A -85,B 0,C 180,E1 -6203.481,E2 -6203.481} C_VEL
LIN {X 0,Y 495.106,Z 548.812,A -85,B 0,C 180,E1 -6204.706,E2 -6204.706} C_VEL
LIN {X 0,Y 495.033,Z 552.427,A -85,B 0,C 180,E1 -6205.93,E2 -6205.93} C_VEL
LIN {X 0,Y 495.042,Z 554.292,A -85,B 0,C 180,E1 -6206.745,E2 -6206.745} C_VEL
LIN {X 0,Y 494.998,Z 555.689,A -85,B 0,C 180,E1 -6207.559,E2 -6207.559} C_VEL
LIN {X 0,Y 494.962,Z 556.685,A -85,B 0,C 180,E1 -6208.373,E2 -6208.373} C_VEL
LIN {X 0,Y 494.901,Z 557.505,A -85,B 0,C 180,E1 -6210,E2 -6210} C_VEL
LIN {X 0,Y 494.962,Z 556.678,A -85,B 0,C 180,E1 -6211.628,E2 -6211.628} C_VEL
LIN {X 0,Y 494.998,Z 555.68,A -85,B 0,C 180,E1 -6212.442,E2 -6212.442} C_VEL
LIN {X 0,Y 495.042,Z 554.28,A -85,B 0,C 180,E1 -6213.256,E2 -6213.256} C_VEL
LIN {X 0,Y 495.008,Z 551.331,A -85,B 0,C 180,E1 -6214.479,E2 -6214.479} C_VEL
LIN {X 0,Y 495.126,Z 547.347,A -85,B 0,C 180,E1 -6215.703,E2 -6215.703} C_VEL
LIN {X 0,Y 495.256,Z 541.218,A -85,B 0,C 180,E1 -6217.133,E2 -6217.133} C_VEL
LIN {X 0,Y 495.422,Z 534.52,A -85,B 0,C 180,E1 -6218.361,E2 -6218.361} C_VEL
LIN {X 0,Y 495.677,Z 526.214,A -85,B 0,C 180,E1 -6219.59,E2 -6219.59} C_VEL
LIN {X 0,Y 495.984,Z 517.701,A -85,B 0,C 180,E1 -6220.615,E2 -6220.615} C_VEL
LIN {X 0,Y 496.436,Z 507.187,A -85,B 0,C 180,E1 -6221.639,E2 -6221.639} C_VEL
LIN {X 0,Y 496.786,Z 495.664,A -85,B 0,C 180,E1 -6222.541,E2 -6222.541} C_VEL
LIN {X 0,Y 497.173,Z 483.459,A -85,B 0,C 180,E1 -6223.28,E2 -6223.28} C_VEL
LIN {X 0,Y 497.561,Z 471.089,A -85,B 0,C 180,E1 -6223.842,E2 -6223.842} C_VEL
LIN {X 0,Y 497.845,Z 458.388,A -85,B 0,C 180,E1 -6224.251,E2 -6224.251} C_VEL
LIN {X 0,Y 498.053,Z 443.299,A -85,B 0,C 180,E1 -6224.532,E2 -6224.532} C_VEL
LIN {X 0,Y 498.476,Z 359.102,A -85,B 0,C 180,E1 -6225.753,E2 -6225.753} C_VEL
LIN {X 0,Y 496.244,Z 344.503,A -85,B 0,C 180,E1 -6226.046,E2 -6226.046} C_VEL
LIN {X 0,Y 496.81,Z 324.929,A -85,B 0,C 180,E1 -6229.202,E2 -6229.202} C_VEL
LIN {X 0,Y 497.482,Z 305.264,A -85,B 0,C 180,E1 -6232.423,E2 -6232.423} C_VEL
LIN {X 0,Y 497.648,Z 298.84,A -85,B 0,C 180,E1 -6233.491,E2 -6233.491} C_VEL
LIN {X 0,Y 495.814,Z 288.726,A -85,B 0,C 180,E1 -6235.306,E2 -6235.306} C_VEL
LIN {X 0,Y 495.781,Z 288.734,A -85,B 0,C 180,E1 -6237.891,E2 -6237.891} C_VEL
LIN {X 0,Y 495.754,Z 288.732,A -85,B 0,C 180,E1 -6240.687,E2 -6240.687} C_VEL
LIN {X 0,Y 495.761,Z 288.727,A -85,B 0,C 180,E1 -6243.564,E2 -6243.564} C_VEL
LIN {X 0,Y 495.729,Z 288.737,A -85,B 0,C 180,E1 -6246.544,E2 -6246.544} C_VEL
LIN {X 0,Y 495.757,Z 288.728,A -85,B 0,C 180,E1 -6249.638,E2 -6249.638} C_VEL
LIN {X 0,Y 495.738,Z 288.736,A -85,B 0,C 180,E1 -6252.507,E2 -6252.507} C_VEL
LIN {X 0,Y 495.738,Z 288.731,A -85,B 0,C 180,E1 -6255.141,E2 -6255.141} C_VEL
LIN {X 0,Y 495.756,Z 288.729,A -85,B 0,C 180,E1 -6258.219,E2 -6258.219} C_VEL
LIN {X 0,Y 495.75,Z 288.728,A -85,B 0,C 180,E1 -6261.408,E2 -6261.408} C_VEL
LIN {X 0,Y 495.747,Z 288.73,A -85,B 0,C 180,E1 -6264.462,E2 -6264.462} C_VEL
LIN {X 0,Y 495.767,Z 288.728,A -85,B 0,C 180,E1 -6267.405,E2 -6267.405} C_VEL
LIN {X 0,Y 495.765,Z 288.724,A -85,B 0,C 180,E1 -6270.253,E2 -6270.253} C_VEL
LIN {X 0,Y 495.823,Z 288.724,A -85,B 0,C 180,E1 -6273.251,E2 -6273.251} C_VEL
LIN {X 0,Y 495.747,Z 288.729,A -85,B 0,C 180,E1 -6275.725,E2 -6275.725} C_VEL
LIN {X 0,Y 495.741,Z 288.727,A -85,B 0,C 180,E1 -6278.371,E2 -6278.371} C_VEL
LIN {X 0,Y 495.783,Z 288.725,A -85,B 0,C 180,E1 -6280.971,E2 -6280.971} C_VEL
LIN {X 0,Y 495.778,Z 288.731,A -85,B 0,C 180,E1 -6283.53,E2 -6283.53} C_VEL
LIN {X 0,Y 495.796,Z 288.722,A -85,B 0,C 180,E1 -6286.056,E2 -6286.056} C_VEL
LIN {X 0,Y 495.849,Z 288.713,A -85,B 0,C 180,E1 -6288.555,E2 -6288.555} C_VEL
LIN {X 0,Y 495.871,Z 288.718,A -85,B 0,C 180,E1 -6291.852,E2 -6291.852} C_VEL
LIN {X 0,Y 495.892,Z 288.707,A -85,B 0,C 180,E1 -6294.306,E2 -6294.306} C_VEL
LIN {X 0,Y 495.991,Z 288.699,A -85,B 0,C 180,E1 -6297.564,E2 -6297.564} C_VEL
LIN {X 0,Y 495.981,Z 288.697,A -85,B 0,C 180,E1 -6300.812,E2 -6300.812} C_VEL
LIN {X 0,Y 495.991,Z 288.697,A -85,B 0,C 180,E1 -6302.436,E2 -6302.436} C_VEL
LIN {X 0,Y 495.887,Z 288.711,A -85,B 0,C 180,E1 -6305.693,E2 -6305.693} C_VEL
LIN {X 0,Y 495.871,Z 288.716,A -85,B 0,C 180,E1 -6308.148,E2 -6308.148} C_VEL
LIN {X 0,Y 495.849,Z 288.713,A -85,B 0,C 180,E1 -6311.445,E2 -6311.445} C_VEL
LIN {X 0,Y 495.792,Z 288.726,A -85,B 0,C 180,E1 -6314.783,E2 -6314.783} C_VEL
LIN {X 0,Y 495.796,Z 288.724,A -85,B 0,C 180,E1 -6318.171,E2 -6318.171} C_VEL
LIN {X 0,Y 495.772,Z 288.73,A -85,B 0,C 180,E1 -6320.756,E2 -6320.756} C_VEL
LIN {X 0,Y 495.75,Z 288.727,A -85,B 0,C 180,E1 -6323.387,E2 -6323.387} C_VEL
LIN {X 0,Y 495.789,Z 288.722,A -85,B 0,C 180,E1 -6326.068,E2 -6326.068} C_VEL
LIN {X 0,Y 495.77,Z 288.729,A -85,B 0,C 180,E1 -6328.815,E2 -6328.815} C_VEL
LIN {X 0,Y 495.753,Z 288.725,A -85,B 0,C 180,E1 -6331.725,E2 -6331.725} C_VEL
LIN {X 0,Y 495.767,Z 288.727,A -85,B 0,C 180,E1 -6334.694,E2 -6334.694} C_VEL
LIN {X 0,Y 495.728,Z 288.733,A -85,B 0,C 180,E1 -6337.562,E2 -6337.562} C_VEL
LIN {X 0,Y 495.765,Z 288.725,A -85,B 0,C 180,E1 -6340.7,E2 -6340.7} C_VEL
LIN {X 0,Y 495.727,Z 288.732,A -85,B 0,C 180,E1 -6344.002,E2 -6344.002} C_VEL
LIN {X 0,Y 495.725,Z 288.734,A -85,B 0,C 180,E1 -6347.117,E2 -6347.117} C_VEL
LIN {X 0,Y 495.758,Z 288.732,A -85,B 0,C 180,E1 -6349.953,E2 -6349.953} C_VEL
LIN {X 0,Y 495.728,Z 288.731,A -85,B 0,C 180,E1 -6352.553,E2 -6352.553} C_VEL
LIN {X 0,Y 495.778,Z 288.729,A -85,B 0,C 180,E1 -6355.457,E2 -6355.457} C_VEL
LIN {X 0,Y 495.756,Z 288.734,A -85,B 0,C 180,E1 -6358.364,E2 -6358.364} C_VEL
LIN {X 0,Y 495.768,Z 288.733,A -85,B 0,C 180,E1 -6359.52,E2 -6359.52} C_VEL
LIN {X 0,Y 495.498,Z 289.424,A -85,B 0,C 180,E1 -6359.968,E2 -6359.968} C_VEL
LIN {X 0,Y 494.57,Z 291.652,A -85,B 0,C 180,E1 -6360.483,E2 -6360.483} C_VEL
LIN {X 0,Y 490.508,Z 300.005,A -85,B 0,C 180,E1 -6361.874,E2 -6361.874} C_VEL
LIN {X 0,Y 489.507,Z 303.204,A -85,B 0,C 180,E1 -6362.45,E2 -6362.45} C_VEL
LIN {X 0,Y 489.405,Z 304.255,A -85,B 0,C 180,E1 -6362.647,E2 -6362.647} C_VEL
LIN {X 0,Y 489.309,Z 310.076,A -85,B 0,C 180,E1 -6363.747,E2 -6363.747} C_VEL
LIN {X 0,Y 491.86,Z 323.325,A -85,B 0,C 180,E1 -6364.056,E2 -6364.056} C_VEL
LIN {X 0,Y 491.141,Z 417.213,A -85,B 0,C 180,E1 -6365.454,E2 -6365.454} C_VEL
LIN {X 0,Y 490.861,Z 430.959,A -85,B 0,C 180,E1 -6365.833,E2 -6365.833} C_VEL
LIN {X 0,Y 490.638,Z 443.505,A -85,B 0,C 180,E1 -6366.354,E2 -6366.354} C_VEL
LIN {X 0,Y 490.26,Z 455.578,A -85,B 0,C 180,E1 -6367.037,E2 -6367.037} C_VEL
LIN {X 0,Y 489.779,Z 467.048,A -85,B 0,C 180,E1 -6367.872,E2 -6367.872} C_VEL
LIN {X 0,Y 489.411,Z 477.71,A -85,B 0,C 180,E1 -6368.851,E2 -6368.851} C_VEL
LIN {X 0,Y 489.02,Z 486.314,A -85,B 0,C 180,E1 -6369.823,E2 -6369.823} C_VEL
LIN {X 0,Y 488.783,Z 494.194,A -85,B 0,C 180,E1 -6370.906,E2 -6370.906} C_VEL
LIN {X 0,Y 488.452,Z 501.077,A -85,B 0,C 180,E1 -6372.054,E2 -6372.054} C_VEL
LIN {X 0,Y 488.243,Z 506.983,A -85,B 0,C 180,E1 -6373.268,E2 -6373.268} C_VEL
LIN {X 0,Y 488.101,Z 512.548,A -85,B 0,C 180,E1 -6374.733,E2 -6374.733} C_VEL
LIN {X 0,Y 488.003,Z 515.685,A -85,B 0,C 180,E1 -6375.828,E2 -6375.828} C_VEL
LIN {X 0,Y 487.919,Z 517.608,A -85,B 0,C 180,E1 -6376.675,E2 -6376.675} C_VEL
LIN {X 0,Y 487.873,Z 519.052,A -85,B 0,C 180,E1 -6377.521,E2 -6377.521} C_VEL
LIN {X 0,Y 487.928,Z 520.063,A -85,B 0,C 180,E1 -6378.366,E2 -6378.366} C_VEL
LIN {X 0,Y 487.884,Z 520.679,A -85,B 0,C 180,E1 -6379.206,E2 -6379.206} C_VEL
LIN {X 0,Y 487.867,Z 520.898,A -85,B 0,C 180,E1 -6380.045,E2 -6380.045} C_VEL
LIN {X 0,Y 487.909,Z 520.057,A -85,B 0,C 180,E1 -6381.718,E2 -6381.718} C_VEL
LIN {X 0,Y 487.925,Z 519.055,A -85,B 0,C 180,E1 -6382.551,E2 -6382.551} C_VEL
LIN {X 0,Y 488.028,Z 517.3,A -85,B 0,C 180,E1 -6383.543,E2 -6383.543} C_VEL
LIN {X 0,Y 487.999,Z 513.492,A -85,B 0,C 180,E1 -6385.043,E2 -6385.043} C_VEL
LIN {X 0,Y 488.178,Z 509.162,A -85,B 0,C 180,E1 -6386.285,E2 -6386.285} C_VEL
LIN {X 0,Y 488.315,Z 503.674,A -85,B 0,C 180,E1 -6387.525,E2 -6387.525} C_VEL
LIN {X 0,Y 488.581,Z 496.835,A -85,B 0,C 180,E1 -6388.763,E2 -6388.763} C_VEL
LIN {X 0,Y 488.93,Z 488.284,A -85,B 0,C 180,E1 -6390,E2 -6390} C_VEL
LIN {X 0,Y 489.207,Z 479.563,A -85,B 0,C 180,E1 -6391.028,E2 -6391.028} C_VEL
LIN {X 0,Y 489.619,Z 468.836,A -85,B 0,C 180,E1 -6392.056,E2 -6392.056} C_VEL
LIN {X 0,Y 490.154,Z 457.983,A -85,B 0,C 180,E1 -6392.876,E2 -6392.876} C_VEL
LIN {X 0,Y 490.515,Z 445.917,A -85,B 0,C 180,E1 -6393.593,E2 -6393.593} C_VEL
LIN {X 0,Y 490.847,Z 433.239,A -85,B 0,C 180,E1 -6394.156,E2 -6394.156} C_VEL
LIN {X 0,Y 491.076,Z 422.631,A -85,B 0,C 180,E1 -6394.488,E2 -6394.488} C_VEL
LIN {X 0,Y 491.215,Z 409.582,A -85,B 0,C 180,E1 -6394.744,E2 -6394.744} C_VEL
LIN {X 0,Y 491.742,Z 323.069,A -85,B 0,C 180,E1 -6396.013,E2 -6396.013} C_VEL
LIN {X 0,Y 489.254,Z 310.215,A -85,B 0,C 180,E1 -6396.288,E2 -6396.288} C_VEL
LIN {X 0,Y 489.513,Z 296.805,A -85,B 0,C 180,E1 -6398.878,E2 -6398.878} C_VEL
LIN {X 0,Y 489.266,Z 292.562,A -85,B 0,C 180,E1 -6399.716,E2 -6399.716} C_VEL
LIN {X 0,Y 488.72,Z 289.611,A -85,B 0,C 180,E1 -6400.355,E2 -6400.355} C_VEL
LIN {X 0,Y 488.736,Z 289.609,A -85,B 0,C 180,E1 -6402.456,E2 -6402.456} C_VEL
LIN {X 0,Y 488.756,Z 289.6,A -85,B 0,C 180,E1 -6405.855,E2 -6405.855} C_VEL
LIN {X 0,Y 488.725,Z 289.602,A -85,B 0,C 180,E1 -6409.313,E2 -6409.313} C_VEL
LIN {X 0,Y 488.695,Z 289.607,A -85,B 0,C 180,E1 -6411.956,E2 -6411.956} C_VEL
LIN {X 0,Y 488.693,Z 289.608,A -85,B 0,C 180,E1 -6415.04,E2 -6415.04} C_VEL
LIN {X 0,Y 488.69,Z 289.61,A -85,B 0,C 180,E1 -6418.331,E2 -6418.331} C_VEL
LIN {X 0,Y 488.681,Z 289.61,A -85,B 0,C 180,E1 -6421.18,E2 -6421.18} C_VEL
LIN {X 0,Y 488.719,Z 289.603,A -85,B 0,C 180,E1 -6424.113,E2 -6424.113} C_VEL
LIN {X 0,Y 488.674,Z 289.613,A -85,B 0,C 180,E1 -6427.158,E2 -6427.158} C_VEL
LIN {X 0,Y 488.687,Z 289.607,A -85,B 0,C 180,E1 -6430.34,E2 -6430.34} C_VEL
LIN {X 0,Y 488.67,Z 289.61,A -85,B 0,C 180,E1 -6433.655,E2 -6433.655} C_VEL
LIN {X 0,Y 488.67,Z 289.609,A -85,B 0,C 180,E1 -6436.344,E2 -6436.344} C_VEL
LIN {X 0,Y 488.696,Z 289.608,A -85,B 0,C 180,E1 -6439.673,E2 -6439.673} C_VEL
LIN {X 0,Y 488.671,Z 289.611,A -85,B 0,C 180,E1 -6442.84,E2 -6442.84} C_VEL
LIN {X 0,Y 488.722,Z 289.604,A -85,B 0,C 180,E1 -6445.887,E2 -6445.887} C_VEL
LIN {X 0,Y 488.683,Z 289.608,A -85,B 0,C 180,E1 -6448.82,E2 -6448.82} C_VEL
LIN {X 0,Y 488.732,Z 289.608,A -85,B 0,C 180,E1 -6451.67,E2 -6451.67} C_VEL
LIN {X 0,Y 488.715,Z 289.603,A -85,B 0,C 180,E1 -6454.443,E2 -6454.443} C_VEL
LIN {X 0,Y 488.713,Z 289.605,A -85,B 0,C 180,E1 -6457.153,E2 -6457.153} C_VEL
LIN {X 0,Y 488.716,Z 289.612,A -85,B 0,C 180,E1 -6459.81,E2 -6459.81} C_VEL
LIN {X 0,Y 488.724,Z 289.603,A -85,B 0,C 180,E1 -6462.423,E2 -6462.423} C_VEL
LIN {X 0,Y 488.752,Z 289.598,A -85,B 0,C 180,E1 -6464.999,E2 -6464.999} C_VEL
LIN {X 0,Y 488.796,Z 289.596,A -85,B 0,C 180,E1 -6468.387,E2 -6468.387} C_VEL
LIN {X 0,Y 488.808,Z 289.595,A -85,B 0,C 180,E1 -6471.734,E2 -6471.734} C_VEL
LIN {X 0,Y 488.798,Z 289.593,A -85,B 0,C 180,E1 -6475.051,E2 -6475.051} C_VEL
LIN {X 0,Y 488.951,Z 289.574,A -85,B 0,C 180,E1 -6477.529,E2 -6477.529} C_VEL
LIN {X 0,Y 488.946,Z 289.577,A -85,B 0,C 180,E1 -6480.824,E2 -6480.824} C_VEL
LIN {X 0,Y 488.951,Z 289.581,A -85,B 0,C 180,E1 -6482.472,E2 -6482.472} C_VEL
LIN {X 0,Y 488.846,Z 289.587,A -85,B 0,C 180,E1 -6485.776,E2 -6485.776} C_VEL
LIN {X 0,Y 488.81,Z 289.596,A -85,B 0,C 180,E1 -6488.267,E2 -6488.267} C_VEL
LIN {X 0,Y 488.799,Z 289.592,A -85,B 0,C 180,E1 -6491.613,E2 -6491.613} C_VEL
LIN {X 0,Y 488.756,Z 289.603,A -85,B 0,C 180,E1 -6495.001,E2 -6495.001} C_VEL
LIN {X 0,Y 488.747,Z 289.603,A -85,B 0,C 180,E1 -6498.443,E2 -6498.443} C_VEL
LIN {X 0,Y 488.699,Z 289.611,A -85,B 0,C 180,E1 -6501.071,E2 -6501.071} C_VEL
LIN {X 0,Y 488.685,Z 289.607,A -85,B 0,C 180,E1 -6503.746,E2 -6503.746} C_VEL
LIN {X 0,Y 488.792,Z 289.601,A -85,B 0,C 180,E1 -6506.946,E2 -6506.946} C_VEL
LIN {X 0,Y 488.712,Z 289.604,A -85,B 0,C 180,E1 -6510.365,E2 -6510.365} C_VEL
LIN {X 0,Y 488.729,Z 289.606,A -85,B 0,C 180,E1 -6513.485,E2 -6513.485} C_VEL
LIN {X 0,Y 488.682,Z 289.607,A -85,B 0,C 180,E1 -6516.356,E2 -6516.356} C_VEL
LIN {X 0,Y 488.697,Z 289.613,A -85,B 0,C 180,E1 -6519.255,E2 -6519.255} C_VEL
LIN {X 0,Y 488.719,Z 289.609,A -85,B 0,C 180,E1 -6521.603,E2 -6521.603} C_VEL
LIN {X 0,Y 488.708,Z 289.605,A -85,B 0,C 180,E1 -6524.802,E2 -6524.802} C_VEL
LIN {X 0,Y 488.688,Z 289.614,A -85,B 0,C 180,E1 -6527.475,E2 -6527.475} C_VEL
LIN {X 0,Y 488.729,Z 289.61,A -85,B 0,C 180,E1 -6529.677,E2 -6529.677} C_VEL
LIN {X 0,Y 488.676,Z 289.608,A -85,B 0,C 180,E1 -6532.842,E2 -6532.842} C_VEL
LIN {X 0,Y 488.728,Z 289.609,A -85,B 0,C 180,E1 -6535.888,E2 -6535.888} C_VEL
LIN {X 0,Y 488.69,Z 289.606,A -85,B 0,C 180,E1 -6538.821,E2 -6538.821} C_VEL
LIN {X 0,Y 488.744,Z 289.607,A -85,B 0,C 180,E1 -6541.672,E2 -6541.672} C_VEL
LIN {X 0,Y 488.798,Z 289.743,A -85,B 0,C 180,E1 -6544.613,E2 -6544.613} C_VEL
LIN {X 0,Y 490.663,Z 300.08,A -85,B 0,C 180,E1 -6546.449,E2 -6546.449} C_VEL
LIN {X 0,Y 490.057,Z 319.363,A -85,B 0,C 180,E1 -6549.65,E2 -6549.65} C_VEL
LIN {X 0,Y 489.412,Z 337.776,A -85,B 0,C 180,E1 -6552.665,E2 -6552.665} C_VEL
LIN {X 0,Y 489.262,Z 344.34,A -85,B 0,C 180,E1 -6553.735,E2 -6553.735} C_VEL
LIN {X 0,Y 491.625,Z 361.064,A -85,B 0,C 180,E1 -6554.065,E2 -6554.065} C_VEL
LIN {X 0,Y 491.041,Z 453.484,A -85,B 0,C 180,E1 -6555.443,E2 -6555.443} C_VEL
LIN {X 0,Y 490.729,Z 467.301,A -85,B 0,C 180,E1 -6555.83,E2 -6555.83} C_VEL
LIN {X 0,Y 490.376,Z 479.161,A -85,B 0,C 180,E1 -6556.322,E2 -6556.322} C_VEL
LIN {X 0,Y 490.016,Z 490.647,A -85,B 0,C 180,E1 -6556.962,E2 -6556.962} C_VEL
LIN {X 0,Y 489.548,Z 502.031,A -85,B 0,C 180,E1 -6557.776,E2 -6557.776} C_VEL
LIN {X 0,Y 489.16,Z 512.508,A -85,B 0,C 180,E1 -6558.712,E2 -6558.712} C_VEL
LIN {X 0,Y 488.835,Z 521.075,A -85,B 0,C 180,E1 -6559.648,E2 -6559.648} C_VEL
LIN {X 0,Y 488.526,Z 528.979,A -85,B 0,C 180,E1 -6560.687,E2 -6560.687} C_VEL
LIN {X 0,Y 488.276,Z 536.7,A -85,B 0,C 180,E1 -6561.933,E2 -6561.933} C_VEL
LIN {X 0,Y 488.073,Z 543.813,A -85,B 0,C 180,E1 -6563.386,E2 -6563.386} C_VEL
LIN {X 0,Y 488.018,Z 548.548,A -85,B 0,C 180,E1 -6564.629,E2 -6564.629} C_VEL
LIN {X 0,Y 487.928,Z 552.162,A -85,B 0,C 180,E1 -6565.871,E2 -6565.871} C_VEL
LIN {X 0,Y 487.964,Z 554.029,A -85,B 0,C 180,E1 -6566.698,E2 -6566.698} C_VEL
LIN {X 0,Y 487.89,Z 556.422,A -85,B 0,C 180,E1 -6568.35,E2 -6568.35} C_VEL
LIN {X 0,Y 487.822,Z 557.242,A -85,B 0,C 180,E1 -6570,E2 -6570} C_VEL
LIN {X 0,Y 487.89,Z 556.414,A -85,B 0,C 180,E1 -6571.651,E2 -6571.651} C_VEL
LIN {X 0,Y 487.965,Z 554.014,A -85,B 0,C 180,E1 -6573.303,E2 -6573.303} C_VEL
LIN {X 0,Y 487.92,Z 551.064,A -85,B 0,C 180,E1 -6574.544,E2 -6574.544} C_VEL
LIN {X 0,Y 488.023,Z 547.077,A -85,B 0,C 180,E1 -6575.786,E2 -6575.786} C_VEL
LIN {X 0,Y 488.182,Z 540.948,A -85,B 0,C 180,E1 -6577.237,E2 -6577.237} C_VEL
LIN {X 0,Y 488.353,Z 534.252,A -85,B 0,C 180,E1 -6578.483,E2 -6578.483} C_VEL
LIN {X 0,Y 488.647,Z 525.949,A -85,B 0,C 180,E1 -6579.73,E2 -6579.73} C_VEL
LIN {X 0,Y 488.992,Z 517.442,A -85,B 0,C 180,E1 -6580.769,E2 -6580.769} C_VEL
LIN {X 0,Y 489.455,Z 506.942,A -85,B 0,C 180,E1 -6581.807,E2 -6581.807} C_VEL
LIN {X 0,Y 489.812,Z 495.603,A -85,B 0,C 180,E1 -6582.71,E2 -6582.71} C_VEL
LIN {X 0,Y 490.245,Z 483.267,A -85,B 0,C 180,E1 -6583.471,E2 -6583.471} C_VEL
LIN {X 0,Y 490.666,Z 470.936,A -85,B 0,C 180,E1 -6584.04,E2 -6584.04} C_VEL
LIN {X 0,Y 490.969,Z 458.302,A -85,B 0,C 180,E1 -6584.455,E2 -6584.455} C_VEL
LIN {X 0,Y 491.182,Z 445.191,A -85,B 0,C 180,E1 -6584.713,E2 -6584.713} C_VEL
LIN {X 0,Y 491.608,Z 359.444,A -85,B 0,C 180,E1 -6585.978,E2 -6585.978} C_VEL
LIN {X 0,Y 489.25,Z 344.18,A -85,B 0,C 180,E1 -6586.299,E2 -6586.299} C_VEL
LIN {X 0,Y 489.818,Z 326.051,A -85,B 0,C 180,E1 -6589.269,E2 -6589.269} C_VEL
LIN {X 0,Y 490.553,Z 306.414,A -85,B 0,C 180,E1 -6592.535,E2 -6592.535} C_VEL
LIN {X 0,Y 490.696,Z 299.865,A -85,B 0,C 180,E1 -6593.643,E2 -6593.643} C_VEL
LIN {X 0,Y 488.789,Z 289.602,A -85,B 0,C 180,E1 -6595.553,E2 -6595.553} C_VEL
LIN {X 0,Y 488.746,Z 289.61,A -85,B 0,C 180,E1 -6598.329,E2 -6598.329} C_VEL
LIN {X 0,Y 488.694,Z 289.61,A -85,B 0,C 180,E1 -6601.18,E2 -6601.18} C_VEL
LIN {X 0,Y 488.732,Z 289.609,A -85,B 0,C 180,E1 -6604.113,E2 -6604.113} C_VEL
LIN {X 0,Y 488.68,Z 289.61,A -85,B 0,C 180,E1 -6607.159,E2 -6607.159} C_VEL
LIN {X 0,Y 488.719,Z 289.61,A -85,B 0,C 180,E1 -6610.344,E2 -6610.344} C_VEL
LIN {X 0,Y 488.685,Z 289.608,A -85,B 0,C 180,E1 -6613.654,E2 -6613.654} C_VEL
LIN {X 0,Y 488.685,Z 289.613,A -85,B 0,C 180,E1 -6616.345,E2 -6616.345} C_VEL
LIN {X 0,Y 488.733,Z 289.6,A -85,B 0,C 180,E1 -6619.676,E2 -6619.676} C_VEL
LIN {X 0,Y 488.679,Z 289.614,A -85,B 0,C 180,E1 -6622.841,E2 -6622.841} C_VEL
LIN {X 0,Y 488.73,Z 289.599,A -85,B 0,C 180,E1 -6625.887,E2 -6625.887} C_VEL
LIN {X 0,Y 488.691,Z 289.612,A -85,B 0,C 180,E1 -6628.82,E2 -6628.82} C_VEL
LIN {X 0,Y 488.744,Z 289.602,A -85,B 0,C 180,E1 -6631.671,E2 -6631.671} C_VEL
LIN {X 0,Y 488.739,Z 289.6,A -85,B 0,C 180,E1 -6634.444,E2 -6634.444} C_VEL
LIN {X 0,Y 488.722,Z 289.608,A -85,B 0,C 180,E1 -6637.153,E2 -6637.153} C_VEL
LIN {X 0,Y 488.724,Z 289.604,A -85,B 0,C 180,E1 -6639.81,E2 -6639.81} C_VEL
LIN {X 0,Y 488.732,Z 289.6,A -85,B 0,C 180,E1 -6642.423,E2 -6642.423} C_VEL
LIN {X 0,Y 488.763,Z 289.598,A -85,B 0,C 180,E1 -6645,E2 -6645} C_VEL
LIN {X 0,Y 488.804,Z 289.591,A -85,B 0,C 180,E1 -6648.387,E2 -6648.387} C_VEL
LIN {X 0,Y 488.815,Z 289.597,A -85,B 0,C 180,E1 -6651.733,E2 -6651.733} C_VEL
LIN {X 0,Y 488.852,Z 289.585,A -85,B 0,C 180,E1 -6654.224,E2 -6654.224} C_VEL
LIN {X 0,Y 488.959,Z 289.574,A -85,B 0,C 180,E1 -6657.529,E2 -6657.529} C_VEL
LIN {X 0,Y 488.932,Z 289.575,A -85,B 0,C 180,E1 -6660.824,E2 -6660.824} C_VEL
LIN {X 0,Y 488.959,Z 289.572,A -85,B 0,C 180,E1 -6662.471,E2 -6662.471} C_VEL
LIN {X 0,Y 488.845,Z 289.589,A -85,B 0,C 180,E1 -6665.776,E2 -6665.776} C_VEL
LIN {X 0,Y 488.815,Z 289.595,A -85,B 0,C 180,E1 -6668.266,E2 -6668.266} C_VEL
LIN {X 0,Y 488.803,Z 289.591,A -85,B 0,C 180,E1 -6671.612,E2 -6671.612} C_VEL
LIN {X 0,Y 488.763,Z 289.599,A -85,B 0,C 180,E1 -6675,E2 -6675} C_VEL
LIN {X 0,Y 488.753,Z 289.605,A -85,B 0,C 180,E1 -6678.442,E2 -6678.442} C_VEL
LIN {X 0,Y 488.705,Z 289.607,A -85,B 0,C 180,E1 -6681.071,E2 -6681.071} C_VEL
LIN {X 0,Y 488.691,Z 289.605,A -85,B 0,C 180,E1 -6683.745,E2 -6683.745} C_VEL
LIN {X 0,Y 488.79,Z 289.6,A -85,B 0,C 180,E1 -6686.944,E2 -6686.944} C_VEL
LIN {X 0,Y 488.708,Z 289.605,A -85,B 0,C 180,E1 -6690.363,E2 -6690.363} C_VEL
LIN {X 0,Y 488.733,Z 289.603,A -85,B 0,C 180,E1 -6693.484,E2 -6693.484} C_VEL
LIN {X 0,Y 488.681,Z 289.608,A -85,B 0,C 180,E1 -6696.355,E2 -6696.355} C_VEL
LIN {X 0,Y 488.7,Z 289.613,A -85,B 0,C 180,E1 -6699.254,E2 -6699.254} C_VEL
LIN {X 0,Y 488.706,Z 289.61,A -85,B 0,C 180,E1 -6701.6,E2 -6701.6} C_VEL
LIN {X 0,Y 488.7,Z 289.607,A -85,B 0,C 180,E1 -6704.803,E2 -6704.803} C_VEL
LIN {X 0,Y 488.691,Z 289.615,A -85,B 0,C 180,E1 -6707.475,E2 -6707.475} C_VEL
LIN {X 0,Y 488.733,Z 289.609,A -85,B 0,C 180,E1 -6709.677,E2 -6709.677} C_VEL
LIN {X 0,Y 488.679,Z 289.609,A -85,B 0,C 180,E1 -6712.841,E2 -6712.841} C_VEL
LIN {X 0,Y 488.731,Z 289.61,A -85,B 0,C 180,E1 -6715.887,E2 -6715.887} C_VEL
LIN {X 0,Y 488.697,Z 289.611,A -85,B 0,C 180,E1 -6718.821,E2 -6718.821} C_VEL
LIN {X 0,Y 488.767,Z 289.762,A -85,B 0,C 180,E1 -6719.843,E2 -6719.843} C_VEL
LIN {X 0,Y 489.525,Z 294.46,A -85,B 0,C 180,E1 -6720.782,E2 -6720.782} C_VEL
LIN {X 0,Y 489.405,Z 304.255,A -85,B 0,C 180,E1 -6722.647,E2 -6722.647} C_VEL
LIN {X 0,Y 489.172,Z 306.714,A -85,B 0,C 180,E1 -6722.995,E2 -6722.995} C_VEL
LIN {X 0,Y 488.675,Z 309.774,A -85,B 0,C 180,E1 -6723.27,E2 -6723.27} C_VEL
LIN {X 0,Y 487.649,Z 315.041,A -85,B 0,C 180,E1 -6723.564,E2 -6723.564} C_VEL
LIN {X 0,Y 486.504,Z 320.877,A -85,B 0,C 180,E1 -6723.749,E2 -6723.749} C_VEL
LIN {X 0,Y 485.81,Z 324.934,A -85,B 0,C 180,E1 -6723.833,E2 -6723.833} C_VEL
LIN {X 0,Y 485.009,Z 333.179,A -85,B 0,C 180,E1 -6723.955,E2 -6723.955} C_VEL
LIN {X 0,Y 484.327,Z 417.351,A -85,B 0,C 180,E1 -6725.228,E2 -6725.228} C_VEL
LIN {X 0,Y 484.046,Z 430.34,A -85,B 0,C 180,E1 -6725.585,E2 -6725.585} C_VEL
LIN {X 0,Y 483.777,Z 442.83,A -85,B 0,C 180,E1 -6726.099,E2 -6726.099} C_VEL
LIN {X 0,Y 483.397,Z 455.398,A -85,B 0,C 180,E1 -6726.807,E2 -6726.807} C_VEL
LIN {X 0,Y 482.879,Z 466.914,A -85,B 0,C 180,E1 -6727.652,E2 -6727.652} C_VEL
LIN {X 0,Y 482.469,Z 477.648,A -85,B 0,C 180,E1 -6728.643,E2 -6728.643} C_VEL
LIN {X 0,Y 482.019,Z 487.157,A -85,B 0,C 180,E1 -6729.74,E2 -6729.74} C_VEL
LIN {X 0,Y 481.673,Z 496.326,A -85,B 0,C 180,E1 -6731.056,E2 -6731.056} C_VEL
LIN {X 0,Y 481.36,Z 503.596,A -85,B 0,C 180,E1 -6732.365,E2 -6732.365} C_VEL
LIN {X 0,Y 481.109,Z 510.15,A -85,B 0,C 180,E1 -6733.886,E2 -6733.886} C_VEL
LIN {X 0,Y 480.988,Z 514.419,A -85,B 0,C 180,E1 -6735.185,E2 -6735.185} C_VEL
LIN {X 0,Y 480.841,Z 517.567,A -85,B 0,C 180,E1 -6736.475,E2 -6736.475} C_VEL
LIN {X 0,Y 480.796,Z 519.116,A -85,B 0,C 180,E1 -6737.334,E2 -6737.334} C_VEL
LIN {X 0,Y 480.841,Z 520.307,A -85,B 0,C 180,E1 -6738.315,E2 -6738.315} C_VEL
LIN {X 0,Y 480.774,Z 521.141,A -85,B 0,C 180,E1 -6739.897,E2 -6739.897} C_VEL
LIN {X 0,Y 480.75,Z 521.02,A -85,B 0,C 180,E1 -6740.746,E2 -6740.746} C_VEL
LIN {X 0,Y 480.806,Z 520.458,A -85,B 0,C 180,E1 -6741.595,E2 -6741.595} C_VEL
LIN {X 0,Y 480.942,Z 518.163,A -85,B 0,C 180,E1 -6743.286,E2 -6743.286} C_VEL
LIN {X 0,Y 480.983,Z 515.333,A -85,B 0,C 180,E1 -6744.55,E2 -6744.55} C_VEL
LIN {X 0,Y 481.049,Z 511.493,A -85,B 0,C 180,E1 -6745.81,E2 -6745.81} C_VEL
LIN {X 0,Y 481.157,Z 506.543,A -85,B 0,C 180,E1 -6747.069,E2 -6747.069} C_VEL
LIN {X 0,Y 481.398,Z 500.331,A -85,B 0,C 180,E1 -6748.326,E2 -6748.326} C_VEL
LIN {X 0,Y 481.77,Z 492.56,A -85,B 0,C 180,E1 -6749.582,E2 -6749.582} C_VEL
LIN {X 0,Y 482.143,Z 482.914,A -85,B 0,C 180,E1 -6750.835,E2 -6750.835} C_VEL
LIN {X 0,Y 482.485,Z 472.93,A -85,B 0,C 180,E1 -6751.878,E2 -6751.878} C_VEL
LIN {X 0,Y 483.113,Z 461.581,A -85,B 0,C 180,E1 -6752.814,E2 -6752.814} C_VEL
LIN {X 0,Y 483.49,Z 450.513,A -85,B 0,C 180,E1 -6753.541,E2 -6753.541} C_VEL
LIN {X 0,Y 483.853,Z 438.098,A -85,B 0,C 180,E1 -6754.164,E2 -6754.164} C_VEL
LIN {X 0,Y 484.087,Z 425.771,A -85,B 0,C 180,E1 -6754.605,E2 -6754.605} C_VEL
LIN {X 0,Y 484.297,Z 413.302,A -85,B 0,C 180,E1 -6754.89,E2 -6754.89} C_VEL
LIN {X 0,Y 484.847,Z 323.462,A -85,B 0,C 180,E1 -6756.231,E2 -6756.231} C_VEL
LIN {X 0,Y 482.295,Z 310.318,A -85,B 0,C 180,E1 -6756.536,E2 -6756.536} C_VEL
LIN {X 0,Y 482.551,Z 297.635,A -85,B 0,C 180,E1 -6759.007,E2 -6759.007} C_VEL
LIN {X 0,Y 482.016,Z 292.325,A -85,B 0,C 180,E1 -6760.076,E2 -6760.076} C_VEL
LIN {X 0,Y 481.691,Z 290.486,A -85,B 0,C 180,E1 -6760.455,E2 -6760.455} C_VEL
LIN {X 0,Y 481.68,Z 290.486,A -85,B 0,C 180,E1 -6762.641,E2 -6762.641} C_VEL
LIN {X 0,Y 481.723,Z 290.475,A -85,B 0,C 180,E1 -6765.657,E2 -6765.657} C_VEL
LIN {X 0,Y 481.702,Z 290.481,A -85,B 0,C 180,E1 -6768.721,E2 -6768.721} C_VEL
LIN {X 0,Y 481.643,Z 290.484,A -85,B 0,C 180,E1 -6771.394,E2 -6771.394} C_VEL
LIN {X 0,Y 481.644,Z 290.487,A -85,B 0,C 180,E1 -6774.114,E2 -6774.114} C_VEL
LIN {X 0,Y 481.648,Z 290.486,A -85,B 0,C 180,E1 -6777.116,E2 -6777.116} C_VEL
LIN {X 0,Y 481.661,Z 290.482,A -85,B 0,C 180,E1 -6779.741,E2 -6779.741} C_VEL
LIN {X 0,Y 481.665,Z 290.489,A -85,B 0,C 180,E1 -6782.674,E2 -6782.674} C_VEL
LIN {X 0,Y 481.631,Z 290.486,A -85,B 0,C 180,E1 -6785.709,E2 -6785.709} C_VEL
LIN {X 0,Y 481.661,Z 290.49,A -85,B 0,C 180,E1 -6788.859,E2 -6788.859} C_VEL
LIN {X 0,Y 481.623,Z 290.486,A -85,B 0,C 180,E1 -6792.162,E2 -6792.162} C_VEL
LIN {X 0,Y 481.647,Z 290.487,A -85,B 0,C 180,E1 -6795.541,E2 -6795.541} C_VEL
LIN {X 0,Y 481.642,Z 290.489,A -85,B 0,C 180,E1 -6798.957,E2 -6798.957} C_VEL
LIN {X 0,Y 481.645,Z 290.484,A -85,B 0,C 180,E1 -6801.992,E2 -6801.992} C_VEL
LIN {X 0,Y 481.68,Z 290.487,A -85,B 0,C 180,E1 -6805.317,E2 -6805.317} C_VEL
LIN {X 0,Y 481.636,Z 290.485,A -85,B 0,C 180,E1 -6808.311,E2 -6808.311} C_VEL
LIN {X 0,Y 481.688,Z 290.483,A -85,B 0,C 180,E1 -6811.218,E2 -6811.218} C_VEL
LIN {X 0,Y 481.675,Z 290.483,A -85,B 0,C 180,E1 -6814.041,E2 -6814.041} C_VEL
LIN {X 0,Y 481.665,Z 290.481,A -85,B 0,C 180,E1 -6816.812,E2 -6816.812} C_VEL
LIN {X 0,Y 481.686,Z 290.484,A -85,B 0,C 180,E1 -6819.502,E2 -6819.502} C_VEL
LIN {X 0,Y 481.698,Z 290.481,A -85,B 0,C 180,E1 -6822.158,E2 -6822.158} C_VEL
LIN {X 0,Y 481.733,Z 290.473,A -85,B 0,C 180,E1 -6824.776,E2 -6824.776} C_VEL
LIN {X 0,Y 481.741,Z 290.477,A -85,B 0,C 180,E1 -6828.215,E2 -6828.215} C_VEL
LIN {X 0,Y 481.753,Z 290.473,A -85,B 0,C 180,E1 -6831.612,E2 -6831.612} C_VEL
LIN {X 0,Y 481.768,Z 290.469,A -85,B 0,C 180,E1 -6834.979,E2 -6834.979} C_VEL
LIN {X 0,Y 481.918,Z 290.45,A -85,B 0,C 180,E1 -6837.493,E2 -6837.493} C_VEL
LIN {X 0,Y 481.897,Z 290.455,A -85,B 0,C 180,E1 -6840.836,E2 -6840.836} C_VEL
LIN {X 0,Y 481.918,Z 290.457,A -85,B 0,C 180,E1 -6842.508,E2 -6842.508} C_VEL
LIN {X 0,Y 481.807,Z 290.465,A -85,B 0,C 180,E1 -6845.861,E2 -6845.861} C_VEL
LIN {X 0,Y 481.756,Z 290.477,A -85,B 0,C 180,E1 -6848.389,E2 -6848.389} C_VEL
LIN {X 0,Y 481.744,Z 290.471,A -85,B 0,C 180,E1 -6851.785,E2 -6851.785} C_VEL
LIN {X 0,Y 481.736,Z 290.475,A -85,B 0,C 180,E1 -6855.225,E2 -6855.225} C_VEL
LIN {X 0,Y 481.704,Z 290.484,A -85,B 0,C 180,E1 -6858.722,E2 -6858.722} C_VEL
LIN {X 0,Y 481.638,Z 290.487,A -85,B 0,C 180,E1 -6861.395,E2 -6861.395} C_VEL
LIN {X 0,Y 481.669,Z 290.481,A -85,B 0,C 180,E1 -6864.114,E2 -6864.114} C_VEL
LIN {X 0,Y 481.745,Z 290.479,A -85,B 0,C 180,E1 -6867.141,E2 -6867.141} C_VEL
LIN {X 0,Y 481.681,Z 290.48,A -85,B 0,C 180,E1 -6869.741,E2 -6869.741} C_VEL
LIN {X 0,Y 481.667,Z 290.483,A -85,B 0,C 180,E1 -6872.675,E2 -6872.675} C_VEL
LIN {X 0,Y 481.636,Z 290.488,A -85,B 0,C 180,E1 -6875.71,E2 -6875.71} C_VEL
LIN {X 0,Y 481.666,Z 290.483,A -85,B 0,C 180,E1 -6878.86,E2 -6878.86} C_VEL
LIN {X 0,Y 481.658,Z 290.485,A -85,B 0,C 180,E1 -6881.915,E2 -6881.915} C_VEL
LIN {X 0,Y 481.656,Z 290.482,A -85,B 0,C 180,E1 -6884.458,E2 -6884.458} C_VEL
LIN {X 0,Y 481.644,Z 290.489,A -85,B 0,C 180,E1 -6887.84,E2 -6887.84} C_VEL
LIN {X 0,Y 481.658,Z 290.482,A -85,B 0,C 180,E1 -6890.655,E2 -6890.655} C_VEL
LIN {X 0,Y 481.624,Z 290.49,A -85,B 0,C 180,E1 -6893.377,E2 -6893.377} C_VEL
LIN {X 0,Y 481.708,Z 290.478,A -85,B 0,C 180,E1 -6896.331,E2 -6896.331} C_VEL
LIN {X 0,Y 481.649,Z 290.486,A -85,B 0,C 180,E1 -6899.418,E2 -6899.418} C_VEL
LIN {X 0,Y 481.7,Z 290.486,A -85,B 0,C 180,E1 -6902.169,E2 -6902.169} C_VEL
LIN {X 0,Y 481.763,Z 290.512,A -85,B 0,C 180,E1 -6904.424,E2 -6904.424} C_VEL
LIN {X 0,Y 483.647,Z 300.764,A -85,B 0,C 180,E1 -6906.273,E2 -6906.273} C_VEL
LIN {X 0,Y 483.212,Z 315.025,A -85,B 0,C 180,E1 -6908.679,E2 -6908.679} C_VEL
LIN {X 0,Y 482.608,Z 333.485,A -85,B 0,C 180,E1 -6911.755,E2 -6911.755} C_VEL
LIN {X 0,Y 482.253,Z 344.145,A -85,B 0,C 180,E1 -6913.512,E2 -6913.512} C_VEL
LIN {X 0,Y 484.761,Z 362.056,A -85,B 0,C 180,E1 -6913.863,E2 -6913.863} C_VEL
LIN {X 0,Y 484.16,Z 452.801,A -85,B 0,C 180,E1 -6915.231,E2 -6915.231} C_VEL
LIN {X 0,Y 483.835,Z 466,A -85,B 0,C 180,E1 -6915.597,E2 -6915.597} C_VEL
LIN {X 0,Y 483.445,Z 478.705,A -85,B 0,C 180,E1 -6916.122,E2 -6916.122} C_VEL
LIN {X 0,Y 483.07,Z 490,A -85,B 0,C 180,E1 -6916.754,E2 -6916.754} C_VEL
LIN {X 0,Y 482.595,Z 501.675,A -85,B 0,C 180,E1 -6917.597,E2 -6917.597} C_VEL
LIN {X 0,Y 482.178,Z 512.179,A -85,B 0,C 180,E1 -6918.546,E2 -6918.546} C_VEL
LIN {X 0,Y 481.816,Z 520.763,A -85,B 0,C 180,E1 -6919.495,E2 -6919.495} C_VEL
LIN {X 0,Y 481.475,Z 528.68,A -85,B 0,C 180,E1 -6920.549,E2 -6920.549} C_VEL
LIN {X 0,Y 481.226,Z 536.415,A -85,B 0,C 180,E1 -6921.814,E2 -6921.814} C_VEL
LIN {X 0,Y 481.005,Z 543.537,A -85,B 0,C 180,E1 -6923.288,E2 -6923.288} C_VEL
LIN {X 0,Y 480.93,Z 548.277,A -85,B 0,C 180,E1 -6924.55,E2 -6924.55} C_VEL
LIN {X 0,Y 480.828,Z 551.893,A -85,B 0,C 180,E1 -6925.809,E2 -6925.809} C_VEL
LIN {X 0,Y 480.888,Z 553.763,A -85,B 0,C 180,E1 -6926.649,E2 -6926.649} C_VEL
LIN {X 0,Y 480.821,Z 556.158,A -85,B 0,C 180,E1 -6928.325,E2 -6928.325} C_VEL
LIN {X 0,Y 480.745,Z 556.978,A -85,B 0,C 180,E1 -6930,E2 -6930} C_VEL
LIN {X 0,Y 480.821,Z 556.151,A -85,B 0,C 180,E1 -6931.676,E2 -6931.676} C_VEL
LIN {X 0,Y 480.888,Z 553.751,A -85,B 0,C 180,E1 -6933.352,E2 -6933.352} C_VEL
LIN {X 0,Y 480.839,Z 550.802,A -85,B 0,C 180,E1 -6934.611,E2 -6934.611} C_VEL
LIN {X 0,Y 480.926,Z 546.818,A -85,B 0,C 180,E1 -6935.872,E2 -6935.872} C_VEL
LIN {X 0,Y 481.107,Z 540.696,A -85,B 0,C 180,E1 -6937.344,E2 -6937.344} C_VEL
LIN {X 0,Y 481.306,Z 534.009,A -85,B 0,C 180,E1 -6938.608,E2 -6938.608} C_VEL
LIN {X 0,Y 481.593,Z 525.716,A -85,B 0,C 180,E1 -6939.874,E2 -6939.874} C_VEL
LIN {X 0,Y 482.006,Z 517.231,A -85,B 0,C 180,E1 -6940.927,E2 -6940.927} C_VEL
LIN {X 0,Y 482.471,Z 506.758,A -85,B 0,C 180,E1 -6941.981,E2 -6941.981} C_VEL
LIN {X 0,Y 482.869,Z 495.477,A -85,B 0,C 180,E1 -6942.894,E2 -6942.894} C_VEL
LIN {X 0,Y 483.351,Z 483.172,A -85,B 0,C 180,E1 -6943.667,E2 -6943.667} C_VEL
LIN {X 0,Y 483.785,Z 470.908,A -85,B 0,C 180,E1 -6944.244,E2 -6944.244} C_VEL
LIN {X 0,Y 484.117,Z 458.389,A -85,B 0,C 180,E1 -6944.664,E2 -6944.664} C_VEL
LIN {X 0,Y 484.331,Z 445.657,A -85,B 0,C 180,E1 -6944.926,E2 -6944.926} C_VEL
LIN {X 0,Y 484.86,Z 361.391,A -85,B 0,C 180,E1 -6946.186,E2 -6946.186} C_VEL
LIN {X 0,Y 482.254,Z 343.861,A -85,B 0,C 180,E1 -6946.565,E2 -6946.565} C_VEL
LIN {X 0,Y 482.879,Z 325.886,A -85,B 0,C 180,E1 -6949.558,E2 -6949.558} C_VEL
LIN {X 0,Y 483.625,Z 307.583,A -85,B 0,C 180,E1 -6952.65,E2 -6952.65} C_VEL
LIN {X 0,Y 483.767,Z 301.138,A -85,B 0,C 180,E1 -6953.759,E2 -6953.759} C_VEL
LIN {X 0,Y 481.753,Z 290.479,A -85,B 0,C 180,E1 -6955.772,E2 -6955.772} C_VEL
LIN {X 0,Y 481.701,Z 290.484,A -85,B 0,C 180,E1 -6958.781,E2 -6958.781} C_VEL
LIN {X 0,Y 481.659,Z 290.491,A -85,B 0,C 180,E1 -6962.189,E2 -6962.189} C_VEL
LIN {X 0,Y 481.69,Z 290.483,A -85,B 0,C 180,E1 -6964.682,E2 -6964.682} C_VEL
LIN {X 0,Y 481.656,Z 290.488,A -85,B 0,C 180,E1 -6968.007,E2 -6968.007} C_VEL
LIN {X 0,Y 481.657,Z 290.486,A -85,B 0,C 180,E1 -6971.042,E2 -6971.042} C_VEL
LIN {X 0,Y 481.655,Z 290.49,A -85,B 0,C 180,E1 -6974.458,E2 -6974.458} C_VEL
LIN {X 0,Y 481.648,Z 290.484,A -85,B 0,C 180,E1 -6977.839,E2 -6977.839} C_VEL
LIN {X 0,Y 481.661,Z 290.487,A -85,B 0,C 180,E1 -6980.654,E2 -6980.654} C_VEL
LIN {X 0,Y 481.627,Z 290.488,A -85,B 0,C 180,E1 -6983.376,E2 -6983.376} C_VEL
LIN {X 0,Y 481.71,Z 290.475,A -85,B 0,C 180,E1 -6986.33,E2 -6986.33} C_VEL
LIN {X 0,Y 481.65,Z 290.486,A -85,B 0,C 180,E1 -6989.417,E2 -6989.417} C_VEL
LIN {X 0,Y 481.699,Z 290.477,A -85,B 0,C 180,E1 -6992.168,E2 -6992.168} C_VEL
LIN {X 0,Y 481.712,Z 290.481,A -85,B 0,C 180,E1 -6994.969,E2 -6994.969} C_VEL
LIN {X 0,Y 481.648,Z 290.487,A -85,B 0,C 180,E1 -6997.705,E2 -6997.705} C_VEL
LIN {X 0,Y 481.704,Z 290.476,A -85,B 0,C 180,E1 -7000.393,E2 -7000.393} C_VEL
LIN {X 0,Y 481.689,Z 290.48,A -85,B 0,C 180,E1 -7003.034,E2 -7003.034} C_VEL
LIN {X 0,Y 481.692,Z 290.482,A -85,B 0,C 180,E1 -7005.639,E2 -7005.639} C_VEL
LIN {X 0,Y 481.749,Z 290.471,A -85,B 0,C 180,E1 -7008.215,E2 -7008.215} C_VEL
LIN {X 0,Y 481.761,Z 290.473,A -85,B 0,C 180,E1 -7011.612,E2 -7011.612} C_VEL
LIN {X 0,Y 481.813,Z 290.463,A -85,B 0,C 180,E1 -7014.139,E2 -7014.139} C_VEL
LIN {X 0,Y 481.926,Z 290.45,A -85,B 0,C 180,E1 -7017.492,E2 -7017.492} C_VEL
LIN {X 0,Y 481.884,Z 290.453,A -85,B 0,C 180,E1 -7020.836,E2 -7020.836} C_VEL
LIN {X 0,Y 481.926,Z 290.448,A -85,B 0,C 180,E1 -7022.507,E2 -7022.507} C_VEL
LIN {X 0,Y 481.805,Z 290.467,A -85,B 0,C 180,E1 -7025.86,E2 -7025.86} C_VEL
LIN {X 0,Y 481.761,Z 290.474,A -85,B 0,C 180,E1 -7028.388,E2 -7028.388} C_VEL
LIN {X 0,Y 481.749,Z 290.471,A -85,B 0,C 180,E1 -7031.785,E2 -7031.785} C_VEL
LIN {X 0,Y 481.742,Z 290.472,A -85,B 0,C 180,E1 -7035.224,E2 -7035.224} C_VEL
LIN {X 0,Y 481.71,Z 290.483,A -85,B 0,C 180,E1 -7038.722,E2 -7038.722} C_VEL
LIN {X 0,Y 481.644,Z 290.484,A -85,B 0,C 180,E1 -7041.395,E2 -7041.395} C_VEL
LIN {X 0,Y 481.675,Z 290.48,A -85,B 0,C 180,E1 -7044.113,E2 -7044.113} C_VEL
LIN {X 0,Y 481.745,Z 290.474,A -85,B 0,C 180,E1 -7047.139,E2 -7047.139} C_VEL
LIN {X 0,Y 481.677,Z 290.48,A -85,B 0,C 180,E1 -7049.741,E2 -7049.741} C_VEL
LIN {X 0,Y 481.67,Z 290.482,A -85,B 0,C 180,E1 -7052.674,E2 -7052.674} C_VEL
LIN {X 0,Y 481.635,Z 290.487,A -85,B 0,C 180,E1 -7055.71,E2 -7055.71} C_VEL
LIN {X 0,Y 481.67,Z 290.484,A -85,B 0,C 180,E1 -7058.859,E2 -7058.859} C_VEL
LIN {X 0,Y 481.652,Z 290.485,A -85,B 0,C 180,E1 -7061.913,E2 -7061.913} C_VEL
LIN {X 0,Y 481.654,Z 290.484,A -85,B 0,C 180,E1 -7064.458,E2 -7064.458} C_VEL
LIN {X 0,Y 481.647,Z 290.489,A -85,B 0,C 180,E1 -7067.839,E2 -7067.839} C_VEL
LIN {X 0,Y 481.661,Z 290.484,A -85,B 0,C 180,E1 -7070.654,E2 -7070.654} C_VEL
LIN {X 0,Y 481.627,Z 290.492,A -85,B 0,C 180,E1 -7073.376,E2 -7073.376} C_VEL
LIN {X 0,Y 481.71,Z 290.482,A -85,B 0,C 180,E1 -7076.33,E2 -7076.33} C_VEL
LIN {X 0,Y 481.704,Z 290.562,A -85,B 0,C 180,E1 -7079.643,E2 -7079.643} C_VEL
LIN {X 0,Y 482.612,Z 296.783,A -85,B 0,C 180,E1 -7080.897,E2 -7080.897} C_VEL
LIN {X 0,Y 482.386,Z 310.644,A -85,B 0,C 180,E1 -7083.511,E2 -7083.511} C_VEL
LIN {X 0,Y 485.126,Z 325.133,A -85,B 0,C 180,E1 -7083.837,E2 -7083.837} C_VEL
LIN {X 0,Y 485.009,Z 333.179,A -85,B 0,C 180,E1 -7083.955,E2 -7083.955} C_VEL
LIN {X 0,Y 484.272,Z 339.022,A -85,B 0,C 180,E1 -7084.017,E2 -7084.017} C_VEL
LIN {X 0,Y 478.719,Z 358.046,A -85,B 0,C 180,E1 -7084.102,E2 -7084.102} C_VEL
LIN {X 0,Y 477.959,Z 363.89,A -85,B 0,C 180,E1 -7084.164,E2 -7084.164} C_VEL
LIN {X 0,Y 477.509,Z 417.657,A -85,B 0,C 180,E1 -7084.996,E2 -7084.996} C_VEL
LIN {X 0,Y 477.214,Z 430.625,A -85,B 0,C 180,E1 -7085.357,E2 -7085.357} C_VEL
LIN {X 0,Y 476.938,Z 443.688,A -85,B 0,C 180,E1 -7085.908,E2 -7085.908} C_VEL
LIN {X 0,Y 476.536,Z 454.747,A -85,B 0,C 180,E1 -7086.534,E2 -7086.534} C_VEL
LIN {X 0,Y 476.088,Z 465.507,A -85,B 0,C 180,E1 -7087.315,E2 -7087.315} C_VEL
LIN {X 0,Y 475.595,Z 476.515,A -85,B 0,C 180,E1 -7088.319,E2 -7088.319} C_VEL
LIN {X 0,Y 475.132,Z 486.349,A -85,B 0,C 180,E1 -7089.433,E2 -7089.433} C_VEL
LIN {X 0,Y 474.769,Z 494.305,A -85,B 0,C 180,E1 -7090.545,E2 -7090.545} C_VEL
LIN {X 0,Y 474.388,Z 502.013,A -85,B 0,C 180,E1 -7091.874,E2 -7091.874} C_VEL
LIN {X 0,Y 474.145,Z 508.15,A -85,B 0,C 180,E1 -7093.199,E2 -7093.199} C_VEL
LIN {X 0,Y 473.973,Z 513.014,A -85,B 0,C 180,E1 -7094.538,E2 -7094.538} C_VEL
LIN {X 0,Y 473.837,Z 516.58,A -85,B 0,C 180,E1 -7095.834,E2 -7095.834} C_VEL
LIN {X 0,Y 473.712,Z 519.145,A -85,B 0,C 180,E1 -7097.141,E2 -7097.141} C_VEL
LIN {X 0,Y 473.76,Z 520.553,A -85,B 0,C 180,E1 -7098.259,E2 -7098.259} C_VEL
LIN {X 0,Y 473.691,Z 521.38,A -85,B 0,C 180,E1 -7099.744,E2 -7099.744} C_VEL
LIN {X 0,Y 473.653,Z 521.324,A -85,B 0,C 180,E1 -7100.606,E2 -7100.606} C_VEL
LIN {X 0,Y 473.719,Z 520.854,A -85,B 0,C 180,E1 -7101.468,E2 -7101.468} C_VEL
LIN {X 0,Y 473.831,Z 518.665,A -85,B 0,C 180,E1 -7103.185,E2 -7103.185} C_VEL
LIN {X 0,Y 473.917,Z 515.94,A -85,B 0,C 180,E1 -7104.468,E2 -7104.468} C_VEL
LIN {X 0,Y 473.945,Z 512.218,A -85,B 0,C 180,E1 -7105.748,E2 -7105.748} C_VEL
LIN {X 0,Y 474.087,Z 507.386,A -85,B 0,C 180,E1 -7107.025,E2 -7107.025} C_VEL
LIN {X 0,Y 474.322,Z 501.308,A -85,B 0,C 180,E1 -7108.301,E2 -7108.301} C_VEL
LIN {X 0,Y 474.704,Z 493.756,A -85,B 0,C 180,E1 -7109.575,E2 -7109.575} C_VEL
LIN {X 0,Y 475.098,Z 484.297,A -85,B 0,C 180,E1 -7110.847,E2 -7110.847} C_VEL
LIN {X 0,Y 475.496,Z 474.563,A -85,B 0,C 180,E1 -7111.905,E2 -7111.905} C_VEL
LIN {X 0,Y 476.001,Z 463.647,A -85,B 0,C 180,E1 -7112.856,E2 -7112.856} C_VEL
LIN {X 0,Y 476.466,Z 452.971,A -85,B 0,C 180,E1 -7113.594,E2 -7113.594} C_VEL
LIN {X 0,Y 476.899,Z 440.142,A -85,B 0,C 180,E1 -7114.278,E2 -7114.278} C_VEL
LIN {X 0,Y 477.085,Z 427.89,A -85,B 0,C 180,E1 -7114.753,E2 -7114.753} C_VEL
LIN {X 0,Y 477.397,Z 415.043,A -85,B 0,C 180,E1 -7115.067,E2 -7115.067} C_VEL
LIN {X 0,Y 478.063,Z 324.664,A -85,B 0,C 180,E1 -7116.436,E2 -7116.436} C_VEL
LIN {X 0,Y 475.329,Z 310.544,A -85,B 0,C 180,E1 -7116.766,E2 -7116.766} C_VEL
LIN {X 0,Y 475.584,Z 298.451,A -85,B 0,C 180,E1 -7119.14,E2 -7119.14} C_VEL
LIN {X 0,Y 474.954,Z 293.134,A -85,B 0,C 180,E1 -7120.227,E2 -7120.227} C_VEL
LIN {X 0,Y 474.624,Z 291.365,A -85,B 0,C 180,E1 -7120.612,E2 -7120.612} C_VEL
LIN {X 0,Y 474.64,Z 291.361,A -85,B 0,C 180,E1 -7122.832,E2 -7122.832} C_VEL
LIN {X 0,Y 474.678,Z 291.353,A -85,B 0,C 180,E1 -7125.766,E2 -7125.766} C_VEL
LIN {X 0,Y 474.656,Z 291.356,A -85,B 0,C 180,E1 -7129.01,E2 -7129.01} C_VEL
LIN {X 0,Y 474.586,Z 291.363,A -85,B 0,C 180,E1 -7131.728,E2 -7131.728} C_VEL
LIN {X 0,Y 474.622,Z 291.367,A -85,B 0,C 180,E1 -7134.494,E2 -7134.494} C_VEL
LIN {X 0,Y 474.595,Z 291.363,A -85,B 0,C 180,E1 -7137.326,E2 -7137.326} C_VEL
LIN {X 0,Y 474.591,Z 291.365,A -85,B 0,C 180,E1 -7140.23,E2 -7140.23} C_VEL
LIN {X 0,Y 474.62,Z 291.362,A -85,B 0,C 180,E1 -7143.221,E2 -7143.221} C_VEL
LIN {X 0,Y 474.584,Z 291.365,A -85,B 0,C 180,E1 -7146.323,E2 -7146.323} C_VEL
LIN {X 0,Y 474.616,Z 291.361,A -85,B 0,C 180,E1 -7149.547,E2 -7149.547} C_VEL
LIN {X 0,Y 474.582,Z 291.364,A -85,B 0,C 180,E1 -7152.231,E2 -7152.231} C_VEL
LIN {X 0,Y 474.61,Z 291.366,A -85,B 0,C 180,E1 -7155.297,E2 -7155.297} C_VEL
LIN {X 0,Y 474.608,Z 291.36,A -85,B 0,C 180,E1 -7158.213,E2 -7158.213} C_VEL
LIN {X 0,Y 474.602,Z 291.366,A -85,B 0,C 180,E1 -7161.542,E2 -7161.542} C_VEL
LIN {X 0,Y 474.616,Z 291.36,A -85,B 0,C 180,E1 -7164.725,E2 -7164.725} C_VEL
LIN {X 0,Y 474.627,Z 291.362,A -85,B 0,C 180,E1 -7167.787,E2 -7167.787} C_VEL
LIN {X 0,Y 474.613,Z 291.361,A -85,B 0,C 180,E1 -7170.885,E2 -7170.885} C_VEL
LIN {X 0,Y 474.627,Z 291.367,A -85,B 0,C 180,E1 -7173.626,E2 -7173.626} C_VEL
LIN {X 0,Y 474.626,Z 291.358,A -85,B 0,C 180,E1 -7176.641,E2 -7176.641} C_VEL
LIN {X 0,Y 474.646,Z 291.36,A -85,B 0,C 180,E1 -7180.089,E2 -7180.089} C_VEL
LIN {X 0,Y 474.641,Z 291.356,A -85,B 0,C 180,E1 -7182.774,E2 -7182.774} C_VEL
LIN {X 0,Y 474.637,Z 291.359,A -85,B 0,C 180,E1 -7185.421,E2 -7185.421} C_VEL
LIN {X 0,Y 474.695,Z 291.358,A -85,B 0,C 180,E1 -7188.037,E2 -7188.037} C_VEL
LIN {X 0,Y 474.719,Z 291.348,A -85,B 0,C 180,E1 -7191.486,E2 -7191.486} C_VEL
LIN {X 0,Y 474.738,Z 291.345,A -85,B 0,C 180,E1 -7194.904,E2 -7194.904} C_VEL
LIN {X 0,Y 474.885,Z 291.326,A -85,B 0,C 180,E1 -7197.455,E2 -7197.455} C_VEL
LIN {X 0,Y 474.848,Z 291.333,A -85,B 0,C 180,E1 -7200.848,E2 -7200.848} C_VEL
LIN {X 0,Y 474.885,Z 291.332,A -85,B 0,C 180,E1 -7202.545,E2 -7202.545} C_VEL
LIN {X 0,Y 474.77,Z 291.342,A -85,B 0,C 180,E1 -7205.948,E2 -7205.948} C_VEL
LIN {X 0,Y 474.721,Z 291.355,A -85,B 0,C 180,E1 -7208.514,E2 -7208.514} C_VEL
LIN {X 0,Y 474.697,Z 291.35,A -85,B 0,C 180,E1 -7211.963,E2 -7211.963} C_VEL
LIN {X 0,Y 474.692,Z 291.35,A -85,B 0,C 180,E1 -7215.456,E2 -7215.456} C_VEL
LIN {X 0,Y 474.657,Z 291.36,A -85,B 0,C 180,E1 -7219.011,E2 -7219.011} C_VEL
LIN {X 0,Y 474.581,Z 291.364,A -85,B 0,C 180,E1 -7221.729,E2 -7221.729} C_VEL
LIN {X 0,Y 474.652,Z 291.357,A -85,B 0,C 180,E1 -7224.493,E2 -7224.493} C_VEL
LIN {X 0,Y 474.692,Z 291.354,A -85,B 0,C 180,E1 -7227.339,E2 -7227.339} C_VEL
LIN {X 0,Y 474.611,Z 291.364,A -85,B 0,C 180,E1 -7230.814,E2 -7230.814} C_VEL
LIN {X 0,Y 474.632,Z 291.358,A -85,B 0,C 180,E1 -7233.985,E2 -7233.985} C_VEL
LIN {X 0,Y 474.57,Z 291.368,A -85,B 0,C 180,E1 -7236.901,E2 -7236.901} C_VEL
LIN {X 0,Y 474.623,Z 291.363,A -85,B 0,C 180,E1 -7239.648,E2 -7239.648} C_VEL
LIN {X 0,Y 474.631,Z 291.359,A -85,B 0,C 180,E1 -7242.933,E2 -7242.933} C_VEL
LIN {X 0,Y 474.605,Z 291.364,A -85,B 0,C 180,E1 -7245.896,E2 -7245.896} C_VEL
LIN {X 0,Y 474.624,Z 291.36,A -85,B 0,C 180,E1 -7249.042,E2 -7249.042} C_VEL
LIN {X 0,Y 474.607,Z 291.37,A -85,B 0,C 180,E1 -7251.705,E2 -7251.705} C_VEL
LIN {X 0,Y 474.622,Z 291.359,A -85,B 0,C 180,E1 -7254.727,E2 -7254.727} C_VEL
LIN {X 0,Y 474.634,Z 291.365,A -85,B 0,C 180,E1 -7257.789,E2 -7257.789} C_VEL
LIN {X 0,Y 474.623,Z 291.362,A -85,B 0,C 180,E1 -7260.885,E2 -7260.885} C_VEL
LIN {X 0,Y 474.672,Z 291.359,A -85,B 0,C 180,E1 -7263.63,E2 -7263.63} C_VEL
LIN {X 0,Y 474.727,Z 291.487,A -85,B 0,C 180,E1 -7264.268,E2 -7264.268} C_VEL
LIN {X 0,Y 476.714,Z 302.21,A -85,B 0,C 180,E1 -7266.23,E2 -7266.23} C_VEL
LIN {X 0,Y 476.173,Z 318.598,A -85,B 0,C 180,E1 -7269.029,E2 -7269.029} C_VEL
LIN {X 0,Y 475.476,Z 337.055,A -85,B 0,C 180,E1 -7272.14,E2 -7272.14} C_VEL
LIN {X 0,Y 475.254,Z 343.819,A -85,B 0,C 180,E1 -7273.272,E2 -7273.272} C_VEL
LIN {X 0,Y 477.893,Z 362.735,A -85,B 0,C 180,E1 -7273.654,E2 -7273.654} C_VEL
LIN {X 0,Y 477.288,Z 451.924,A -85,B 0,C 180,E1 -7275.013,E2 -7275.013} C_VEL
LIN {X 0,Y 476.994,Z 465.348,A -85,B 0,C 180,E1 -7275.386,E2 -7275.386} C_VEL
LIN {X 0,Y 476.537,Z 478.158,A -85,B 0,C 180,E1 -7275.917,E2 -7275.917} C_VEL
LIN {X 0,Y 476.129,Z 489.541,A -85,B 0,C 180,E1 -7276.558,E2 -7276.558} C_VEL
LIN {X 0,Y 475.666,Z 500.603,A -85,B 0,C 180,E1 -7277.358,E2 -7277.358} C_VEL
LIN {X 0,Y 475.2,Z 511.803,A -85,B 0,C 180,E1 -7278.375,E2 -7278.375} C_VEL
LIN {X 0,Y 474.778,Z 520.409,A -85,B 0,C 180,E1 -7279.338,E2 -7279.338} C_VEL
LIN {X 0,Y 474.447,Z 528.348,A -85,B 0,C 180,E1 -7280.408,E2 -7280.408} C_VEL
LIN {X 0,Y 474.162,Z 536.104,A -85,B 0,C 180,E1 -7281.691,E2 -7281.691} C_VEL
LIN {X 0,Y 473.921,Z 543.238,A -85,B 0,C 180,E1 -7283.187,E2 -7283.187} C_VEL
LIN {X 0,Y 473.844,Z 547.988,A -85,B 0,C 180,E1 -7284.468,E2 -7284.468} C_VEL
LIN {X 0,Y 473.735,Z 551.613,A -85,B 0,C 180,E1 -7285.747,E2 -7285.747} C_VEL
LIN {X 0,Y 473.795,Z 553.487,A -85,B 0,C 180,E1 -7286.599,E2 -7286.599} C_VEL
LIN {X 0,Y 473.741,Z 554.889,A -85,B 0,C 180,E1 -7287.45,E2 -7287.45} C_VEL
LIN {X 0,Y 473.724,Z 555.888,A -85,B 0,C 180,E1 -7288.3,E2 -7288.3} C_VEL
LIN {X 0,Y 473.672,Z 556.714,A -85,B 0,C 180,E1 -7290,E2 -7290} C_VEL
LIN {X 0,Y 473.689,Z 556.499,A -85,B 0,C 180,E1 -7290.851,E2 -7290.851} C_VEL
LIN {X 0,Y 473.724,Z 555.891,A -85,B 0,C 180,E1 -7291.701,E2 -7291.701} C_VEL
LIN {X 0,Y 473.795,Z 553.497,A -85,B 0,C 180,E1 -7293.402,E2 -7293.402} C_VEL
LIN {X 0,Y 473.762,Z 550.554,A -85,B 0,C 180,E1 -7294.68,E2 -7294.68} C_VEL
LIN {X 0,Y 473.833,Z 546.576,A -85,B 0,C 180,E1 -7295.96,E2 -7295.96} C_VEL
LIN {X 0,Y 474.016,Z 540.469,A -85,B 0,C 180,E1 -7297.454,E2 -7297.454} C_VEL
LIN {X 0,Y 474.254,Z 533.795,A -85,B 0,C 180,E1 -7298.737,E2 -7298.737} C_VEL
LIN {X 0,Y 474.559,Z 525.52,A -85,B 0,C 180,E1 -7300.021,E2 -7300.021} C_VEL
LIN {X 0,Y 475.018,Z 517.063,A -85,B 0,C 180,E1 -7301.09,E2 -7301.09} C_VEL
LIN {X 0,Y 475.498,Z 506.819,A -85,B 0,C 180,E1 -7302.141,E2 -7302.141} C_VEL
LIN {X 0,Y 475.931,Z 495.031,A -85,B 0,C 180,E1 -7303.112,E2 -7303.112} C_VEL
LIN {X 0,Y 476.445,Z 483.161,A -85,B 0,C 180,E1 -7303.869,E2 -7303.869} C_VEL
LIN {X 0,Y 476.922,Z 470.989,A -85,B 0,C 180,E1 -7304.454,E2 -7304.454} C_VEL
LIN {X 0,Y 477.304,Z 457.722,A -85,B 0,C 180,E1 -7304.905,E2 -7304.905} C_VEL
LIN {X 0,Y 477.511,Z 444.634,A -85,B 0,C 180,E1 -7305.171,E2 -7305.171} C_VEL
LIN {X 0,Y 478.076,Z 362.238,A -85,B 0,C 180,E1 -7306.422,E2 -7306.422} C_VEL
LIN {X 0,Y 475.292,Z 343.535,A -85,B 0,C 180,E1 -7306.842,E2 -7306.842} C_VEL
LIN {X 0,Y 476.048,Z 324.437,A -85,B 0,C 180,E1 -7310.075,E2 -7310.075} C_VEL
LIN {X 0,Y 476.815,Z 306.159,A -85,B 0,C 180,E1 -7313.221,E2 -7313.221} C_VEL
LIN {X 0,Y 476.648,Z 301.241,A -85,B 0,C 180,E1 -7314.099,E2 -7314.099} C_VEL
LIN {X 0,Y 474.7,Z 291.358,A -85,B 0,C 180,E1 -7316.014,E2 -7316.014} C_VEL
LIN {X 0,Y 474.647,Z 291.367,A -85,B 0,C 180,E1 -7318.282,E2 -7318.282} C_VEL
LIN {X 0,Y 474.601,Z 291.366,A -85,B 0,C 180,E1 -7321.218,E2 -7321.218} C_VEL
LIN {X 0,Y 474.634,Z 291.367,A -85,B 0,C 180,E1 -7324.241,E2 -7324.241} C_VEL
LIN {X 0,Y 474.591,Z 291.365,A -85,B 0,C 180,E1 -7327.384,E2 -7327.384} C_VEL
LIN {X 0,Y 474.618,Z 291.367,A -85,B 0,C 180,E1 -7330.658,E2 -7330.658} C_VEL
LIN {X 0,Y 474.601,Z 291.363,A -85,B 0,C 180,E1 -7333.481,E2 -7333.481} C_VEL
LIN {X 0,Y 474.601,Z 291.37,A -85,B 0,C 180,E1 -7336.519,E2 -7336.519} C_VEL
LIN {X 0,Y 474.617,Z 291.36,A -85,B 0,C 180,E1 -7339.342,E2 -7339.342} C_VEL
LIN {X 0,Y 474.59,Z 291.369,A -85,B 0,C 180,E1 -7342.616,E2 -7342.616} C_VEL
LIN {X 0,Y 474.631,Z 291.356,A -85,B 0,C 180,E1 -7345.759,E2 -7345.759} C_VEL
LIN {X 0,Y 474.598,Z 291.367,A -85,B 0,C 180,E1 -7348.782,E2 -7348.782} C_VEL
LIN {X 0,Y 474.645,Z 291.357,A -85,B 0,C 180,E1 -7351.717,E2 -7351.717} C_VEL
LIN {X 0,Y 474.652,Z 291.356,A -85,B 0,C 180,E1 -7354.582,E2 -7354.582} C_VEL
LIN {X 0,Y 474.6,Z 291.367,A -85,B 0,C 180,E1 -7357.355,E2 -7357.355} C_VEL
LIN {X 0,Y 474.653,Z 291.355,A -85,B 0,C 180,E1 -7360.089,E2 -7360.089} C_VEL
LIN {X 0,Y 474.649,Z 291.355,A -85,B 0,C 180,E1 -7362.774,E2 -7362.774} C_VEL
LIN {X 0,Y 474.65,Z 291.359,A -85,B 0,C 180,E1 -7365.421,E2 -7365.421} C_VEL
LIN {X 0,Y 474.702,Z 291.35,A -85,B 0,C 180,E1 -7368.037,E2 -7368.037} C_VEL
LIN {X 0,Y 474.726,Z 291.348,A -85,B 0,C 180,E1 -7371.486,E2 -7371.486} C_VEL
LIN {X 0,Y 474.776,Z 291.34,A -85,B 0,C 180,E1 -7374.052,E2 -7374.052} C_VEL
LIN {X 0,Y 474.892,Z 291.326,A -85,B 0,C 180,E1 -7377.455,E2 -7377.455} C_VEL
LIN {X 0,Y 474.909,Z 291.326,A -85,B 0,C 180,E1 -7380,E2 -7380} C_VEL
LIN {X 0,Y 474.892,Z 291.323,A -85,B 0,C 180,E1 -7382.545,E2 -7382.545} C_VEL
LIN {X 0,Y 474.768,Z 291.344,A -85,B 0,C 180,E1 -7385.948,E2 -7385.948} C_VEL
LIN {X 0,Y 474.726,Z 291.35,A -85,B 0,C 180,E1 -7388.513,E2 -7388.513} C_VEL
LIN {X 0,Y 474.702,Z 291.35,A -85,B 0,C 180,E1 -7391.962,E2 -7391.962} C_VEL
